LIN {X 0,Y 520,Z 902.665,A -85,B 0,C 180,E1 12177.794,E2 12177.794} C_VEL
LIN {X 0,Y 524.952,Z 869.378,A -85,B 0,C 180,E1 12181.307,E2 12181.307} C_VEL
LIN {X 0,Y 530.595,Z 831.105,A -85,B 0,C 180,E1 12184.398,E2 12184.398} C_VEL
LIN {X 0,Y 536.264,Z 787.905,A -85,B 0,C 180,E1 12186.977,E2 12186.977} C_VEL
LIN {X 0,Y 540.929,Z 743.185,A -85,B 0,C 180,E1 12188.852,E2 12188.852} C_VEL
LIN {X 0,Y 544.188,Z 696.094,A -85,B 0,C 180,E1 12190.101,E2 12190.101} C_VEL
LIN {X 0,Y 544.022,Z 681.132,A -85,B 0,C 180,E1 12190.406,E2 12190.406} C_VEL
LIN {X 0,Y 507.953,Z 601.31,A -85,B 0,C 180,E1 12194.386,E2 12194.386} C_VEL
LIN {X 0,Y 507.831,Z 601.31,A -85,B 0,C 180,E1 12200.881,E2 12200.881} C_VEL
LIN {X 0,Y 507.959,Z 601.31,A -85,B 0,C 180,E1 12206.647,E2 12206.647} C_VEL
LIN {X 0,Y 508.168,Z 601.31,A -85,B 0,C 180,E1 12211.51,E2 12211.51} C_VEL
LIN {X 0,Y 508.405,Z 601.31,A -85,B 0,C 180,E1 12217.515,E2 12217.515} C_VEL
LIN {X 0,Y 508.487,Z 601.31,A -85,B 0,C 180,E1 12222.665,E2 12222.665} C_VEL
LIN {X 0,Y 508.666,Z 601.31,A -85,B 0,C 180,E1 12227.965,E2 12227.965} C_VEL
LIN {X 0,Y 508.95,Z 601.31,A -85,B 0,C 180,E1 12233.16,E2 12233.16} C_VEL
LIN {X 0,Y 509.131,Z 601.31,A -85,B 0,C 180,E1 12238.293,E2 12238.293} C_VEL
LIN {X 0,Y 509.118,Z 601.31,A -85,B 0,C 180,E1 12243.41,E2 12243.41} C_VEL
LIN {X 0,Y 508.825,Z 601.31,A -85,B 0,C 180,E1 12248.559,E2 12248.559} C_VEL
LIN {X 0,Y 508.651,Z 601.31,A -85,B 0,C 180,E1 12253.782,E2 12253.782} C_VEL
LIN {X 0,Y 508.481,Z 601.31,A -85,B 0,C 180,E1 12259.128,E2 12259.128} C_VEL
LIN {X 0,Y 508.251,Z 601.31,A -85,B 0,C 180,E1 12264.661,E2 12264.661} C_VEL
LIN {X 0,Y 508.106,Z 601.31,A -85,B 0,C 180,E1 12270.451,E2 12270.451} C_VEL
LIN {X 0,Y 507.956,Z 601.31,A -85,B 0,C 180,E1 12276.614,E2 12276.614} C_VEL
LIN {X 0,Y 507.883,Z 601.31,A -85,B 0,C 180,E1 12283.314,E2 12283.314} C_VEL
LIN {X 0,Y 507.816,Z 601.31,A -85,B 0,C 180,E1 12288.966,E2 12288.966} C_VEL
LIN {X 0,Y 508.01,Z 601.31,A -85,B 0,C 180,E1 12295.314,E2 12295.314} C_VEL
LIN {X 0,Y 528.495,Z 651.414,A -85,B 0,C 180,E1 12298.224,E2 12298.224} C_VEL
LIN {X 0,Y 532.04,Z 668.727,A -85,B 0,C 180,E1 12299.099,E2 12299.099} C_VEL
LIN {X 0,Y 528.891,Z 707.618,A -85,B 0,C 180,E1 12300.849,E2 12300.849} C_VEL
LIN {X 0,Y 525.082,Z 743.156,A -85,B 0,C 180,E1 12303.155,E2 12303.155} C_VEL
LIN {X 0,Y 521.047,Z 775.217,A -85,B 0,C 180,E1 12305.971,E2 12305.971} C_VEL
LIN {X 0,Y 517.204,Z 804.444,A -85,B 0,C 180,E1 12309.413,E2 12309.413} C_VEL
LIN {X 0,Y 514.215,Z 827.771,A -85,B 0,C 180,E1 12313.102,E2 12313.102} C_VEL
LIN {X 0,Y 512.171,Z 846.045,A -85,B 0,C 180,E1 12317.034,E2 12317.034} C_VEL
LIN {X 0,Y 511.03,Z 859.031,A -85,B 0,C 180,E1 12321.04,E2 12321.04} C_VEL
LIN {X 0,Y 510.473,Z 866.812,A -85,B 0,C 180,E1 12324.887,E2 12324.887} C_VEL
LIN {X 0,Y 510.207,Z 870.137,A -85,B 0,C 180,E1 12328.294,E2 12328.294} C_VEL
LIN {X 0,Y 510.347,Z 870.07,A -85,B 0,C 180,E1 12331.697,E2 12331.697} C_VEL
LIN {X 0,Y 510.589,Z 865.782,A -85,B 0,C 180,E1 12335.703,E2 12335.703} C_VEL
LIN {X 0,Y 511.119,Z 856.498,A -85,B 0,C 180,E1 12339.81,E2 12339.81} C_VEL
LIN {X 0,Y 512.543,Z 842.831,A -85,B 0,C 180,E1 12343.675,E2 12343.675} C_VEL
LIN {X 0,Y 514.927,Z 822.28,A -85,B 0,C 180,E1 12347.771,E2 12347.771} C_VEL
LIN {X 0,Y 518.198,Z 797.24,A -85,B 0,C 180,E1 12351.433,E2 12351.433} C_VEL
LIN {X 0,Y 522.167,Z 766.734,A -85,B 0,C 180,E1 12354.763,E2 12354.763} C_VEL
LIN {X 0,Y 526.179,Z 733.773,A -85,B 0,C 180,E1 12357.43,E2 12357.43} C_VEL
LIN {X 0,Y 529.775,Z 697.922,A -85,B 0,C 180,E1 12359.557,E2 12359.557} C_VEL
LIN {X 0,Y 531.526,Z 665.249,A -85,B 0,C 180,E1 12360.976,E2 12360.976} C_VEL
LIN {X 0,Y 524.161,Z 639.669,A -85,B 0,C 180,E1 12362.329,E2 12362.329} C_VEL
LIN {X 0,Y 508.103,Z 601.31,A -85,B 0,C 180,E1 12364.601,E2 12364.601} C_VEL
LIN {X 0,Y 507.864,Z 601.31,A -85,B 0,C 180,E1 12371.017,E2 12371.017} C_VEL
LIN {X 0,Y 507.854,Z 601.31,A -85,B 0,C 180,E1 12376.683,E2 12376.683} C_VEL
LIN {X 0,Y 507.918,Z 601.31,A -85,B 0,C 180,E1 12383.383,E2 12383.383} C_VEL
LIN {X 0,Y 508.13,Z 601.31,A -85,B 0,C 180,E1 12389.846,E2 12389.846} C_VEL
LIN {X 0,Y 508.314,Z 601.31,A -85,B 0,C 180,E1 12394.173,E2 12394.173} C_VEL
LIN {X 0,Y 524.583,Z 651.894,A -85,B 0,C 180,E1 12395.94,E2 12395.94} C_VEL
LIN {X 0,Y 522.857,Z 701.074,A -85,B 0,C 180,E1 12396.974,E2 12396.974} C_VEL
LIN {X 0,Y 520.724,Z 738.628,A -85,B 0,C 180,E1 12398.437,E2 12398.437} C_VEL
LIN {X 0,Y 518.128,Z 773.015,A -85,B 0,C 180,E1 12400.466,E2 12400.466} C_VEL
LIN {X 0,Y 515.733,Z 803.731,A -85,B 0,C 180,E1 12403.031,E2 12403.031} C_VEL
LIN {X 0,Y 513.615,Z 830.564,A -85,B 0,C 180,E1 12406.137,E2 12406.137} C_VEL
LIN {X 0,Y 512.062,Z 851.637,A -85,B 0,C 180,E1 12409.562,E2 12409.562} C_VEL
LIN {X 0,Y 511.289,Z 866.871,A -85,B 0,C 180,E1 12413.196,E2 12413.196} C_VEL
LIN {X 0,Y 511.021,Z 875.647,A -85,B 0,C 180,E1 12416.603,E2 12416.603} C_VEL
LIN {X 0,Y 511.016,Z 879.604,A -85,B 0,C 180,E1 12420.002,E2 12420.002} C_VEL
LIN {X 0,Y 511.336,Z 878.832,A -85,B 0,C 180,E1 12423.399,E2 12423.399} C_VEL
LIN {X 0,Y 512.187,Z 873.073,A -85,B 0,C 180,E1 12426.797,E2 12426.797} C_VEL
LIN {X 0,Y 513.564,Z 862.006,A -85,B 0,C 180,E1 12430.196,E2 12430.196} C_VEL
LIN {X 0,Y 515.523,Z 844.762,A -85,B 0,C 180,E1 12433.599,E2 12433.599} C_VEL
LIN {X 0,Y 517.943,Z 822.966,A -85,B 0,C 180,E1 12436.571,E2 12436.571} C_VEL
LIN {X 0,Y 520.985,Z 794.562,A -85,B 0,C 180,E1 12439.378,E2 12439.378} C_VEL
LIN {X 0,Y 524.438,Z 759.753,A -85,B 0,C 180,E1 12441.835,E2 12441.835} C_VEL
LIN {X 0,Y 528.068,Z 719.982,A -85,B 0,C 180,E1 12443.78,E2 12443.78} C_VEL
LIN {X 0,Y 531.717,Z 674.928,A -85,B 0,C 180,E1 12445.188,E2 12445.188} C_VEL
LIN {X 0,Y 532.545,Z 655.359,A -85,B 0,C 180,E1 12445.707,E2 12445.707} C_VEL
LIN {X 0,Y 523.124,Z 630.3,A -85,B 0,C 180,E1 12447.507,E2 12447.507} C_VEL
LIN {X 0,Y 513.846,Z 612.495,A -85,B 0,C 180,E1 12449.435,E2 12449.435} C_VEL
LIN {X 0,Y 510.034,Z 606.45,A -85,B 0,C 180,E1 12450.329,E2 12450.329} C_VEL
LIN {X 0,Y 508.092,Z 601.31,A -85,B 0,C 180,E1 12451.036,E2 12451.036} C_VEL
LIN {X 0,Y 508,Z 601.31,A -85,B 0,C 180,E1 12456.616,E2 12456.616} C_VEL
LIN {X 0,Y 507.909,Z 601.31,A -85,B 0,C 180,E1 12463.317,E2 12463.317} C_VEL
LIN {X 0,Y 507.889,Z 601.868,A -85,B 0,C 180,E1 12464.024,E2 12464.024} C_VEL
LIN {X 0,Y 510.593,Z 607.203,A -85,B 0,C 180,E1 12464.707,E2 12464.707} C_VEL
LIN {X 0,Y 519.408,Z 621.579,A -85,B 0,C 180,E1 12466.437,E2 12466.437} C_VEL
LIN {X 0,Y 530.121,Z 643.576,A -85,B 0,C 180,E1 12468.173,E2 12468.173} C_VEL
LIN {X 0,Y 538.662,Z 670.296,A -85,B 0,C 180,E1 12469.492,E2 12469.492} C_VEL
LIN {X 0,Y 542.514,Z 685.222,A -85,B 0,C 180,E1 12470.096,E2 12470.096} C_VEL
LIN {X 0,Y 539.64,Z 730.719,A -85,B 0,C 180,E1 12471.16,E2 12471.16} C_VEL
LIN {X 0,Y 535.552,Z 773.807,A -85,B 0,C 180,E1 12472.795,E2 12472.795} C_VEL
LIN {X 0,Y 530.748,Z 816.248,A -85,B 0,C 180,E1 12475.111,E2 12475.111} C_VEL
LIN {X 0,Y 525.549,Z 855.463,A -85,B 0,C 180,E1 12477.983,E2 12477.983} C_VEL
LIN {X 0,Y 524.944,Z 859.637,A -85,B 0,C 180,E1 12478.346,E2 12478.346} C_VEL
LIN {X 0,Y 519.28,Z 873.172,A -85,B 0,C 180,E1 12479.413,E2 12479.413} C_VEL
LIN {X 0,Y 513.783,Z 886.061,A -85,B 0,C 180,E1 12480.57,E2 12480.57} C_VEL
LIN {X 0,Y 509.18,Z 917.936,A -85,B 0,C 180,E1 12484.443,E2 12484.443} C_VEL
LIN {X 0,Y 505.687,Z 945.186,A -85,B 0,C 180,E1 12488.724,E2 12488.724} C_VEL
LIN {X 0,Y 503.449,Z 967.671,A -85,B 0,C 180,E1 12493.391,E2 12493.391} C_VEL
LIN {X 0,Y 502.283,Z 984.168,A -85,B 0,C 180,E1 12498.167,E2 12498.167} C_VEL
LIN {X 0,Y 501.854,Z 993.668,A -85,B 0,C 180,E1 12502.196,E2 12502.196} C_VEL
LIN {X 0,Y 501.774,Z 999.535,A -85,B 0,C 180,E1 12506.542,E2 12506.542} C_VEL
LIN {X 0,Y 501.842,Z 1001.106,A -85,B 0,C 180,E1 12510.005,E2 12510.005} C_VEL
LIN {X 0,Y 501.849,Z 998.33,A -85,B 0,C 180,E1 12515.012,E2 12515.012} C_VEL
LIN {X 0,Y 501.97,Z 989.857,A -85,B 0,C 180,E1 12520,E2 12520} C_VEL
LIN {X 0,Y 502.842,Z 976.424,A -85,B 0,C 180,E1 12524.732,E2 12524.732} C_VEL
LIN {X 0,Y 504.859,Z 955.712,A -85,B 0,C 180,E1 12529.738,E2 12529.738} C_VEL
LIN {X 0,Y 508.329,Z 929.158,A -85,B 0,C 180,E1 12534.435,E2 12534.435} C_VEL
LIN {X 0,Y 512.81,Z 899.389,A -85,B 0,C 180,E1 12538.438,E2 12538.438} C_VEL
LIN {X 0,Y 518.058,Z 865.903,A -85,B 0,C 180,E1 12541.928,E2 12541.928} C_VEL
LIN {X 0,Y 523.721,Z 828.076,A -85,B 0,C 180,E1 12544.955,E2 12544.955} C_VEL
LIN {X 0,Y 529.236,Z 787.2,A -85,B 0,C 180,E1 12547.397,E2 12547.397} C_VEL
LIN {X 0,Y 534.129,Z 741.814,A -85,B 0,C 180,E1 12549.31,E2 12549.31} C_VEL
LIN {X 0,Y 537.459,Z 694.943,A -85,B 0,C 180,E1 12550.55,E2 12550.55} C_VEL
LIN {X 0,Y 537.203,Z 683.382,A -85,B 0,C 180,E1 12550.795,E2 12550.795} C_VEL
LIN {X 0,Y 500.024,Z 601.31,A -85,B 0,C 180,E1 12554.978,E2 12554.978} C_VEL
LIN {X 0,Y 499.903,Z 601.31,A -85,B 0,C 180,E1 12560.475,E2 12560.475} C_VEL
LIN {X 0,Y 500.061,Z 601.31,A -85,B 0,C 180,E1 12566.953,E2 12566.953} C_VEL
LIN {X 0,Y 500.242,Z 601.31,A -85,B 0,C 180,E1 12572.981,E2 12572.981} C_VEL
LIN {X 0,Y 500.476,Z 601.31,A -85,B 0,C 180,E1 12578.699,E2 12578.699} C_VEL
LIN {X 0,Y 500.619,Z 601.31,A -85,B 0,C 180,E1 12584.194,E2 12584.194} C_VEL
LIN {X 0,Y 500.847,Z 601.31,A -85,B 0,C 180,E1 12589.542,E2 12589.542} C_VEL
LIN {X 0,Y 501.148,Z 601.31,A -85,B 0,C 180,E1 12594.795,E2 12594.795} C_VEL
LIN {X 0,Y 501.325,Z 601.31,A -85,B 0,C 180,E1 12599.998,E2 12599.998} C_VEL
LIN {X 0,Y 501.177,Z 601.31,A -85,B 0,C 180,E1 12605.201,E2 12605.201} C_VEL
LIN {X 0,Y 500.866,Z 601.31,A -85,B 0,C 180,E1 12610.453,E2 12610.453} C_VEL
LIN {X 0,Y 500.654,Z 601.31,A -85,B 0,C 180,E1 12615.8,E2 12615.8} C_VEL
LIN {X 0,Y 500.499,Z 601.31,A -85,B 0,C 180,E1 12621.295,E2 12621.295} C_VEL
LIN {X 0,Y 500.227,Z 601.31,A -85,B 0,C 180,E1 12627.015,E2 12627.015} C_VEL
LIN {X 0,Y 500.08,Z 601.31,A -85,B 0,C 180,E1 12633.041,E2 12633.041} C_VEL
LIN {X 0,Y 499.942,Z 601.31,A -85,B 0,C 180,E1 12639.515,E2 12639.515} C_VEL
LIN {X 0,Y 499.975,Z 601.31,A -85,B 0,C 180,E1 12645.804,E2 12645.804} C_VEL
LIN {X 0,Y 499.894,Z 601.31,A -85,B 0,C 180,E1 12651.987,E2 12651.987} C_VEL
LIN {X 0,Y 500.05,Z 601.31,A -85,B 0,C 180,E1 12654.652,E2 12654.652} C_VEL
LIN {X 0,Y 520.969,Z 651.493,A -85,B 0,C 180,E1 12657.696,E2 12657.696} C_VEL
LIN {X 0,Y 525.141,Z 671.855,A -85,B 0,C 180,E1 12658.754,E2 12658.754} C_VEL
LIN {X 0,Y 521.749,Z 710.935,A -85,B 0,C 180,E1 12660.575,E2 12660.575} C_VEL
LIN {X 0,Y 517.831,Z 745.962,A -85,B 0,C 180,E1 12662.916,E2 12662.916} C_VEL
LIN {X 0,Y 513.605,Z 778.182,A -85,B 0,C 180,E1 12665.827,E2 12665.827} C_VEL
LIN {X 0,Y 509.516,Z 807.297,A -85,B 0,C 180,E1 12669.376,E2 12669.376} C_VEL
LIN {X 0,Y 506.449,Z 830.412,A -85,B 0,C 180,E1 12673.165,E2 12673.165} C_VEL
LIN {X 0,Y 504.3,Z 848.89,A -85,B 0,C 180,E1 12677.322,E2 12677.322} C_VEL
LIN {X 0,Y 503.139,Z 861.13,A -85,B 0,C 180,E1 12681.335,E2 12681.335} C_VEL
LIN {X 0,Y 502.601,Z 868.987,A -85,B 0,C 180,E1 12685.673,E2 12685.673} C_VEL
LIN {X 0,Y 502.513,Z 871.538,A -85,B 0,C 180,E1 12689.995,E2 12689.995} C_VEL
LIN {X 0,Y 502.633,Z 868.872,A -85,B 0,C 180,E1 12694.317,E2 12694.317} C_VEL
LIN {X 0,Y 503.231,Z 860.902,A -85,B 0,C 180,E1 12698.654,E2 12698.654} C_VEL
LIN {X 0,Y 504.5,Z 847.214,A -85,B 0,C 180,E1 12703.016,E2 12703.016} C_VEL
LIN {X 0,Y 506.733,Z 828.038,A -85,B 0,C 180,E1 12707.19,E2 12707.19} C_VEL
LIN {X 0,Y 510.106,Z 803.151,A -85,B 0,C 180,E1 12711.105,E2 12711.105} C_VEL
LIN {X 0,Y 514.092,Z 774.214,A -85,B 0,C 180,E1 12714.481,E2 12714.481} C_VEL
LIN {X 0,Y 518.385,Z 741.285,A -85,B 0,C 180,E1 12717.351,E2 12717.351} C_VEL
LIN {X 0,Y 522.276,Z 705.207,A -85,B 0,C 180,E1 12719.645,E2 12719.645} C_VEL
LIN {X 0,Y 524.671,Z 667.194,A -85,B 0,C 180,E1 12721.37,E2 12721.37} C_VEL
LIN {X 0,Y 517.609,Z 642.557,A -85,B 0,C 180,E1 12722.713,E2 12722.713} C_VEL
LIN {X 0,Y 500.132,Z 601.31,A -85,B 0,C 180,E1 12725.243,E2 12725.243} C_VEL
LIN {X 0,Y 499.999,Z 601.31,A -85,B 0,C 180,E1 12731.806,E2 12731.806} C_VEL
LIN {X 0,Y 499.941,Z 601.31,A -85,B 0,C 180,E1 12738.196,E2 12738.196} C_VEL
LIN {X 0,Y 500.033,Z 601.31,A -85,B 0,C 180,E1 12744.892,E2 12744.892} C_VEL
LIN {X 0,Y 500.249,Z 601.31,A -85,B 0,C 180,E1 12751.438,E2 12751.438} C_VEL
LIN {X 0,Y 500.361,Z 601.31,A -85,B 0,C 180,E1 12753.777,E2 12753.777} C_VEL
LIN {X 0,Y 517.186,Z 655.212,A -85,B 0,C 180,E1 12755.678,E2 12755.678} C_VEL
LIN {X 0,Y 515.422,Z 701.486,A -85,B 0,C 180,E1 12756.683,E2 12756.683} C_VEL
LIN {X 0,Y 513.224,Z 738.97,A -85,B 0,C 180,E1 12758.166,E2 12758.166} C_VEL
LIN {X 0,Y 510.497,Z 774.133,A -85,B 0,C 180,E1 12760.275,E2 12760.275} C_VEL
LIN {X 0,Y 507.881,Z 805.823,A -85,B 0,C 180,E1 12762.984,E2 12762.984} C_VEL
LIN {X 0,Y 505.767,Z 832.36,A -85,B 0,C 180,E1 12766.138,E2 12766.138} C_VEL
LIN {X 0,Y 504.242,Z 853.261,A -85,B 0,C 180,E1 12769.618,E2 12769.618} C_VEL
LIN {X 0,Y 503.42,Z 868.26,A -85,B 0,C 180,E1 12773.293,E2 12773.293} C_VEL
LIN {X 0,Y 503.198,Z 876.534,A -85,B 0,C 180,E1 12776.55,E2 12776.55} C_VEL
LIN {X 0,Y 503.195,Z 880.651,A -85,B 0,C 180,E1 12780.002,E2 12780.002} C_VEL
LIN {X 0,Y 503.537,Z 880.006,A -85,B 0,C 180,E1 12783.452,E2 12783.452} C_VEL
LIN {X 0,Y 504.456,Z 874.408,A -85,B 0,C 180,E1 12786.901,E2 12786.901} C_VEL
LIN {X 0,Y 505.933,Z 863.428,A -85,B 0,C 180,E1 12790.352,E2 12790.352} C_VEL
LIN {X 0,Y 508.01,Z 846.33,A -85,B 0,C 180,E1 12793.804,E2 12793.804} C_VEL
LIN {X 0,Y 510.587,Z 824.772,A -85,B 0,C 180,E1 12796.817,E2 12796.817} C_VEL
LIN {X 0,Y 513.842,Z 796.322,A -85,B 0,C 180,E1 12799.696,E2 12799.696} C_VEL
LIN {X 0,Y 517.401,Z 762.529,A -85,B 0,C 180,E1 12802.148,E2 12802.148} C_VEL
LIN {X 0,Y 521.217,Z 723.88,A -85,B 0,C 180,E1 12804.127,E2 12804.127} C_VEL
LIN {X 0,Y 524.994,Z 682.276,A -85,B 0,C 180,E1 12805.535,E2 12805.535} C_VEL
LIN {X 0,Y 526.375,Z 657.824,A -85,B 0,C 180,E1 12806.206,E2 12806.206} C_VEL
LIN {X 0,Y 517.228,Z 633.141,A -85,B 0,C 180,E1 12808.099,E2 12808.099} C_VEL
LIN {X 0,Y 507.4,Z 614.083,A -85,B 0,C 180,E1 12810.387,E2 12810.387} C_VEL
LIN {X 0,Y 502.885,Z 607.264,A -85,B 0,C 180,E1 12811.64,E2 12811.64} C_VEL
LIN {X 0,Y 500.132,Z 601.853,A -85,B 0,C 180,E1 12812.655,E2 12812.655} C_VEL
LIN {X 0,Y 499.988,Z 601.31,A -85,B 0,C 180,E1 12818.016,E2 12818.016} C_VEL
LIN {X 0,Y 500.023,Z 601.976,A -85,B 0,C 180,E1 12822.293,E2 12822.293} C_VEL
LIN {X 0,Y 502.726,Z 607.254,A -85,B 0,C 180,E1 12823.217,E2 12823.217} C_VEL
LIN {X 0,Y 504.974,Z 610.344,A -85,B 0,C 180,E1 12823.816,E2 12823.816} C_VEL
LIN {X 0,Y 512.671,Z 622.71,A -85,B 0,C 180,E1 12825.547,E2 12825.547} C_VEL
LIN {X 0,Y 522.833,Z 642.836,A -85,B 0,C 180,E1 12827.38,E2 12827.38} C_VEL
LIN {X 0,Y 530.974,Z 666.365,A -85,B 0,C 180,E1 12828.724,E2 12828.724} C_VEL
LIN {X 0,Y 536.271,Z 685.119,A -85,B 0,C 180,E1 12829.578,E2 12829.578} C_VEL
LIN {X 0,Y 533.213,Z 730.537,A -85,B 0,C 180,E1 12830.665,E2 12830.665} C_VEL
LIN {X 0,Y 528.819,Z 773.973,A -85,B 0,C 180,E1 12832.345,E2 12832.345} C_VEL
LIN {X 0,Y 523.816,Z 815.666,A -85,B 0,C 180,E1 12834.659,E2 12834.659} C_VEL
LIN {X 0,Y 518.24,Z 855.553,A -85,B 0,C 180,E1 12837.635,E2 12837.635} C_VEL
LIN {X 0,Y 513.783,Z 886.061,A -85,B 0,C 180,E1 12840.57,E2 12840.57} C_VEL
LIN {X 0,Y 511.734,Z 892.403,A -85,B 0,C 180,E1 12841.213,E2 12841.213} C_VEL
LIN {X 0,Y 502.927,Z 908.748,A -85,B 0,C 180,E1 12842.967,E2 12842.967} C_VEL
LIN {X 0,Y 502.65,Z 910.185,A -85,B 0,C 180,E1 12843.151,E2 12843.151} C_VEL
LIN {X 0,Y 498.838,Z 937.618,A -85,B 0,C 180,E1 12847.266,E2 12847.266} C_VEL
LIN {X 0,Y 496.197,Z 960.3,A -85,B 0,C 180,E1 12851.654,E2 12851.654} C_VEL
LIN {X 0,Y 494.6,Z 979.493,A -85,B 0,C 180,E1 12856.722,E2 12856.722} C_VEL
LIN {X 0,Y 494.084,Z 990.97,A -85,B 0,C 180,E1 12861.185,E2 12861.185} C_VEL
LIN {X 0,Y 494.027,Z 996.816,A -85,B 0,C 180,E1 12864.726,E2 12864.726} C_VEL
LIN {X 0,Y 494.011,Z 999.798,A -85,B 0,C 180,E1 12868.247,E2 12868.247} C_VEL
LIN {X 0,Y 493.881,Z 999.942,A -85,B 0,C 180,E1 12871.763,E2 12871.763} C_VEL
LIN {X 0,Y 493.93,Z 996.144,A -85,B 0,C 180,E1 12876.168,E2 12876.168} C_VEL
LIN {X 0,Y 494.288,Z 986.415,A -85,B 0,C 180,E1 12881.256,E2 12881.256} C_VEL
LIN {X 0,Y 495.482,Z 970.106,A -85,B 0,C 180,E1 12886.437,E2 12886.437} C_VEL
LIN {X 0,Y 497.803,Z 948.823,A -85,B 0,C 180,E1 12891.194,E2 12891.194} C_VEL
LIN {X 0,Y 501.484,Z 923.247,A -85,B 0,C 180,E1 12895.508,E2 12895.508} C_VEL
LIN {X 0,Y 506.338,Z 892.85,A -85,B 0,C 180,E1 12899.464,E2 12899.464} C_VEL
LIN {X 0,Y 512.022,Z 857.355,A -85,B 0,C 180,E1 12903.018,E2 12903.018} C_VEL
LIN {X 0,Y 518.09,Z 816.765,A -85,B 0,C 180,E1 12906.085,E2 12906.085} C_VEL
LIN {X 0,Y 523.914,Z 771.768,A -85,B 0,C 180,E1 12908.538,E2 12908.538} C_VEL
LIN {X 0,Y 528.471,Z 726.177,A -85,B 0,C 180,E1 12910.225,E2 12910.225} C_VEL
LIN {X 0,Y 530.451,Z 685.946,A -85,B 0,C 180,E1 12911.175,E2 12911.175} C_VEL
LIN {X 0,Y 492.065,Z 601.31,A -85,B 0,C 180,E1 12915.556,E2 12915.556} C_VEL
LIN {X 0,Y 492.01,Z 601.31,A -85,B 0,C 180,E1 12921.988,E2 12921.988} C_VEL
LIN {X 0,Y 492.168,Z 601.31,A -85,B 0,C 180,E1 12928.447,E2 12928.447} C_VEL
LIN {X 0,Y 492.348,Z 601.31,A -85,B 0,C 180,E1 12934.482,E2 12934.482} C_VEL
LIN {X 0,Y 492.582,Z 601.31,A -85,B 0,C 180,E1 12940.225,E2 12940.225} C_VEL
LIN {X 0,Y 492.729,Z 601.31,A -85,B 0,C 180,E1 12945.759,E2 12945.759} C_VEL
LIN {X 0,Y 493.001,Z 601.31,A -85,B 0,C 180,E1 12951.16,E2 12951.16} C_VEL
LIN {X 0,Y 493.338,Z 601.31,A -85,B 0,C 180,E1 12956.477,E2 12956.477} C_VEL
LIN {X 0,Y 493.447,Z 601.31,A -85,B 0,C 180,E1 12961.757,E2 12961.757} C_VEL
LIN {X 0,Y 493.111,Z 601.31,A -85,B 0,C 180,E1 12967.056,E2 12967.056} C_VEL
LIN {X 0,Y 492.847,Z 601.31,A -85,B 0,C 180,E1 12972.423,E2 12972.423} C_VEL
LIN {X 0,Y 492.667,Z 601.31,A -85,B 0,C 180,E1 12977.905,E2 12977.905} C_VEL
LIN {X 0,Y 492.444,Z 601.31,A -85,B 0,C 180,E1 12983.57,E2 12983.57} C_VEL
LIN {X 0,Y 492.227,Z 601.31,A -85,B 0,C 180,E1 12989.497,E2 12989.497} C_VEL
LIN {X 0,Y 492.058,Z 601.31,A -85,B 0,C 180,E1 12995.796,E2 12995.796} C_VEL
LIN {X 0,Y 492.059,Z 601.31,A -85,B 0,C 180,E1 13002.343,E2 13002.343} C_VEL
LIN {X 0,Y 492.036,Z 601.31,A -85,B 0,C 180,E1 13007.636,E2 13007.636} C_VEL
LIN {X 0,Y 492.167,Z 601.598,A -85,B 0,C 180,E1 13014.002,E2 13014.002} C_VEL
LIN {X 0,Y 513.135,Z 650.798,A -85,B 0,C 180,E1 13017.111,E2 13017.111} C_VEL
LIN {X 0,Y 518.412,Z 672.347,A -85,B 0,C 180,E1 13018.302,E2 13018.302} C_VEL
LIN {X 0,Y 514.926,Z 711.698,A -85,B 0,C 180,E1 13020.146,E2 13020.146} C_VEL
LIN {X 0,Y 510.696,Z 747.83,A -85,B 0,C 180,E1 13022.595,E2 13022.595} C_VEL
LIN {X 0,Y 506.301,Z 780.014,A -85,B 0,C 180,E1 13025.561,E2 13025.561} C_VEL
LIN {X 0,Y 502.029,Z 809.024,A -85,B 0,C 180,E1 13029.176,E2 13029.176} C_VEL
LIN {X 0,Y 498.707,Z 832.634,A -85,B 0,C 180,E1 13033.147,E2 13033.147} C_VEL
LIN {X 0,Y 496.459,Z 851.295,A -85,B 0,C 180,E1 13037.528,E2 13037.528} C_VEL
LIN {X 0,Y 495.221,Z 864.071,A -85,B 0,C 180,E1 13042.081,E2 13042.081} C_VEL
LIN {X 0,Y 494.684,Z 870.844,A -85,B 0,C 180,E1 13046.483,E2 13046.483} C_VEL
LIN {X 0,Y 494.675,Z 872.526,A -85,B 0,C 180,E1 13049.995,E2 13049.995} C_VEL
LIN {X 0,Y 494.813,Z 869.855,A -85,B 0,C 180,E1 13054.386,E2 13054.386} C_VEL
LIN {X 0,Y 495.451,Z 861.878,A -85,B 0,C 180,E1 13058.791,E2 13058.791} C_VEL
LIN {X 0,Y 496.831,Z 848.192,A -85,B 0,C 180,E1 13063.216,E2 13063.216} C_VEL
LIN {X 0,Y 499.153,Z 829.396,A -85,B 0,C 180,E1 13067.38,E2 13067.38} C_VEL
LIN {X 0,Y 502.767,Z 804.065,A -85,B 0,C 180,E1 13071.428,E2 13071.428} C_VEL
LIN {X 0,Y 506.928,Z 775.109,A -85,B 0,C 180,E1 13074.85,E2 13074.85} C_VEL
LIN {X 0,Y 511.48,Z 741.669,A -85,B 0,C 180,E1 13077.792,E2 13077.792} C_VEL
LIN {X 0,Y 515.585,Z 704.541,A -85,B 0,C 180,E1 13080.15,E2 13080.15} C_VEL
LIN {X 0,Y 517.838,Z 669.07,A -85,B 0,C 180,E1 13081.776,E2 13081.776} C_VEL
LIN {X 0,Y 510.746,Z 644.586,A -85,B 0,C 180,E1 13083.158,E2 13083.158} C_VEL
LIN {X 0,Y 492.218,Z 601.31,A -85,B 0,C 180,E1 13085.917,E2 13085.917} C_VEL
LIN {X 0,Y 492.059,Z 601.31,A -85,B 0,C 180,E1 13092.638,E2 13092.638} C_VEL
LIN {X 0,Y 492.02,Z 601.31,A -85,B 0,C 180,E1 13097.647,E2 13097.647} C_VEL
LIN {X 0,Y 492.01,Z 601.31,A -85,B 0,C 180,E1 13104.2,E2 13104.2} C_VEL
LIN {X 0,Y 492.242,Z 601.31,A -85,B 0,C 180,E1 13110.504,E2 13110.504} C_VEL
LIN {X 0,Y 492.42,Z 601.31,A -85,B 0,C 180,E1 13113.362,E2 13113.362} C_VEL
LIN {X 0,Y 509.852,Z 655.963,A -85,B 0,C 180,E1 13115.367,E2 13115.367} C_VEL
LIN {X 0,Y 508.001,Z 702.075,A -85,B 0,C 180,E1 13116.389,E2 13116.389} C_VEL
LIN {X 0,Y 505.719,Z 739.812,A -85,B 0,C 180,E1 13117.913,E2 13117.913} C_VEL
LIN {X 0,Y 502.863,Z 775.24,A -85,B 0,C 180,E1 13120.077,E2 13120.077} C_VEL
LIN {X 0,Y 500.286,Z 806.05,A -85,B 0,C 180,E1 13122.746,E2 13122.746} C_VEL
LIN {X 0,Y 498.071,Z 832.625,A -85,B 0,C 180,E1 13125.92,E2 13125.92} C_VEL
LIN {X 0,Y 496.455,Z 853.767,A -85,B 0,C 180,E1 13129.453,E2 13129.453} C_VEL
LIN {X 0,Y 495.677,Z 868.314,A -85,B 0,C 180,E1 13132.98,E2 13132.98} C_VEL
LIN {X 0,Y 495.373,Z 877.429,A -85,B 0,C 180,E1 13136.496,E2 13136.496} C_VEL
LIN {X 0,Y 495.366,Z 881.699,A -85,B 0,C 180,E1 13140.002,E2 13140.002} C_VEL
LIN {X 0,Y 495.741,Z 881.191,A -85,B 0,C 180,E1 13143.506,E2 13143.506} C_VEL
LIN {X 0,Y 496.745,Z 875.739,A -85,B 0,C 180,E1 13147.009,E2 13147.009} C_VEL
LIN {X 0,Y 498.303,Z 864.915,A -85,B 0,C 180,E1 13150.512,E2 13150.512} C_VEL
LIN {X 0,Y 500.521,Z 847.972,A -85,B 0,C 180,E1 13154.014,E2 13154.014} C_VEL
LIN {X 0,Y 503.505,Z 824.841,A -85,B 0,C 180,E1 13157.286,E2 13157.286} C_VEL
LIN {X 0,Y 506.992,Z 795.99,A -85,B 0,C 180,E1 13160.214,E2 13160.214} C_VEL
LIN {X 0,Y 511.097,Z 760.341,A -85,B 0,C 180,E1 13162.793,E2 13162.793} C_VEL
LIN {X 0,Y 515.223,Z 721.295,A -85,B 0,C 180,E1 13164.773,E2 13164.773} C_VEL
LIN {X 0,Y 519.331,Z 678.345,A -85,B 0,C 180,E1 13166.21,E2 13166.21} C_VEL
LIN {X 0,Y 520.369,Z 660.306,A -85,B 0,C 180,E1 13166.736,E2 13166.736} C_VEL
LIN {X 0,Y 511.959,Z 637.259,A -85,B 0,C 180,E1 13168.61,E2 13168.61} C_VEL
LIN {X 0,Y 503.435,Z 620.256,A -85,B 0,C 180,E1 13170.769,E2 13170.769} C_VEL
LIN {X 0,Y 498.729,Z 613.018,A -85,B 0,C 180,E1 13172.215,E2 13172.215} C_VEL
LIN {X 0,Y 496.132,Z 608.125,A -85,B 0,C 180,E1 13173.297,E2 13173.297} C_VEL
LIN {X 0,Y 492.169,Z 602.151,A -85,B 0,C 180,E1 13175.759,E2 13175.759} C_VEL
LIN {X 0,Y 492.075,Z 601.654,A -85,B 0,C 180,E1 13179.032,E2 13179.032} C_VEL
LIN {X 0,Y 495.389,Z 607.746,A -85,B 0,C 180,E1 13181.301,E2 13181.301} C_VEL
LIN {X 0,Y 497.333,Z 609.914,A -85,B 0,C 180,E1 13182.04,E2 13182.04} C_VEL
LIN {X 0,Y 502.656,Z 618.608,A -85,B 0,C 180,E1 13183.712,E2 13183.712} C_VEL
LIN {X 0,Y 510.552,Z 631.664,A -85,B 0,C 180,E1 13185.511,E2 13185.511} C_VEL
LIN {X 0,Y 520.242,Z 653.231,A -85,B 0,C 180,E1 13187.331,E2 13187.331} C_VEL
LIN {X 0,Y 529.915,Z 686.896,A -85,B 0,C 180,E1 13189.055,E2 13189.055} C_VEL
LIN {X 0,Y 526.636,Z 732.845,A -85,B 0,C 180,E1 13190.223,E2 13190.223} C_VEL
LIN {X 0,Y 521.861,Z 776.603,A -85,B 0,C 180,E1 13191.991,E2 13191.991} C_VEL
LIN {X 0,Y 516.652,Z 817.297,A -85,B 0,C 180,E1 13194.335,E2 13194.335} C_VEL
LIN {X 0,Y 511.037,Z 855.396,A -85,B 0,C 180,E1 13197.247,E2 13197.247} C_VEL
LIN {X 0,Y 505.494,Z 891.768,A -85,B 0,C 180,E1 13200.886,E2 13200.886} C_VEL
LIN {X 0,Y 502.65,Z 910.185,A -85,B 0,C 180,E1 13203.151,E2 13203.151} C_VEL
LIN {X 0,Y 500.658,Z 915.879,A -85,B 0,C 180,E1 13203.879,E2 13203.879} C_VEL
LIN {X 0,Y 492.108,Z 930.466,A -85,B 0,C 180,E1 13205.889,E2 13205.889} C_VEL
LIN {X 0,Y 491.865,Z 931.76,A -85,B 0,C 180,E1 13206.093,E2 13206.093} C_VEL
LIN {X 0,Y 488.673,Z 956.569,A -85,B 0,C 180,E1 13210.777,E2 13210.777} C_VEL
LIN {X 0,Y 486.948,Z 975.488,A -85,B 0,C 180,E1 13215.591,E2 13215.591} C_VEL
LIN {X 0,Y 486.282,Z 988.134,A -85,B 0,C 180,E1 13220.137,E2 13220.137} C_VEL
LIN {X 0,Y 486.183,Z 995.909,A -85,B 0,C 180,E1 13224.64,E2 13224.64} C_VEL
LIN {X 0,Y 486.159,Z 998.914,A -85,B 0,C 180,E1 13228.219,E2 13228.219} C_VEL
LIN {X 0,Y 486.033,Z 999.074,A -85,B 0,C 180,E1 13231.791,E2 13231.791} C_VEL
LIN {X 0,Y 486.063,Z 995.249,A -85,B 0,C 180,E1 13236.269,E2 13236.269} C_VEL
LIN {X 0,Y 486.417,Z 985.462,A -85,B 0,C 180,E1 13241.44,E2 13241.44} C_VEL
LIN {X 0,Y 487.659,Z 969.038,A -85,B 0,C 180,E1 13246.708,E2 13246.708} C_VEL
LIN {X 0,Y 490.135,Z 947.596,A -85,B 0,C 180,E1 13251.542,E2 13251.542} C_VEL
LIN {X 0,Y 494.016,Z 921.782,A -85,B 0,C 180,E1 13255.922,E2 13255.922} C_VEL
LIN {X 0,Y 498.937,Z 891.624,A -85,B 0,C 180,E1 13259.871,E2 13259.871} C_VEL
LIN {X 0,Y 504.887,Z 855.882,A -85,B 0,C 180,E1 13263.472,E2 13263.472} C_VEL
LIN {X 0,Y 511.123,Z 815.171,A -85,B 0,C 180,E1 13266.553,E2 13266.553} C_VEL
LIN {X 0,Y 516.91,Z 771.703,A -85,B 0,C 180,E1 13268.945,E2 13268.945} C_VEL
LIN {X 0,Y 521.704,Z 724.989,A -85,B 0,C 180,E1 13270.685,E2 13270.685} C_VEL
LIN {X 0,Y 523.8,Z 688.696,A -85,B 0,C 180,E1 13271.551,E2 13271.551} C_VEL
LIN {X 0,Y 485.425,Z 605.588,A -85,B 0,C 180,E1 13275.906,E2 13275.906} C_VEL
LIN {X 0,Y 484.14,Z 601.31,A -85,B 0,C 180,E1 13276.112,E2 13276.112} C_VEL
LIN {X 0,Y 484.064,Z 601.31,A -85,B 0,C 180,E1 13281.502,E2 13281.502} C_VEL
LIN {X 0,Y 484.175,Z 601.31,A -85,B 0,C 180,E1 13287.864,E2 13287.864} C_VEL
LIN {X 0,Y 484.412,Z 601.31,A -85,B 0,C 180,E1 13294.033,E2 13294.033} C_VEL
LIN {X 0,Y 484.631,Z 601.31,A -85,B 0,C 180,E1 13299.886,E2 13299.886} C_VEL
LIN {X 0,Y 484.824,Z 601.31,A -85,B 0,C 180,E1 13305.677,E2 13305.677} C_VEL
LIN {X 0,Y 485.084,Z 601.31,A -85,B 0,C 180,E1 13311.014,E2 13311.014} C_VEL
LIN {X 0,Y 485.429,Z 601.31,A -85,B 0,C 180,E1 13316.419,E2 13316.419} C_VEL
LIN {X 0,Y 485.541,Z 601.31,A -85,B 0,C 180,E1 13321.786,E2 13321.786} C_VEL
LIN {X 0,Y 485.188,Z 601.31,A -85,B 0,C 180,E1 13327.172,E2 13327.172} C_VEL
LIN {X 0,Y 484.919,Z 601.31,A -85,B 0,C 180,E1 13332.629,E2 13332.629} C_VEL
LIN {X 0,Y 484.72,Z 601.31,A -85,B 0,C 180,E1 13338.209,E2 13338.209} C_VEL
LIN {X 0,Y 484.474,Z 601.31,A -85,B 0,C 180,E1 13343.982,E2 13343.982} C_VEL
LIN {X 0,Y 484.292,Z 601.31,A -85,B 0,C 180,E1 13350.029,E2 13350.029} C_VEL
LIN {X 0,Y 484.12,Z 601.31,A -85,B 0,C 180,E1 13356.477,E2 13356.477} C_VEL
LIN {X 0,Y 484.072,Z 601.31,A -85,B 0,C 180,E1 13361.296,E2 13361.296} C_VEL
LIN {X 0,Y 484.046,Z 601.31,A -85,B 0,C 180,E1 13366.469,E2 13366.469} C_VEL
LIN {X 0,Y 484.175,Z 601.31,A -85,B 0,C 180,E1 13373.242,E2 13373.242} C_VEL
LIN {X 0,Y 505.554,Z 650.75,A -85,B 0,C 180,E1 13376.542,E2 13376.542} C_VEL
LIN {X 0,Y 511.693,Z 673.462,A -85,B 0,C 180,E1 13377.862,E2 13377.862} C_VEL
LIN {X 0,Y 508.086,Z 712.755,A -85,B 0,C 180,E1 13379.721,E2 13379.721} C_VEL
LIN {X 0,Y 503.706,Z 748.879,A -85,B 0,C 180,E1 13382.2,E2 13382.2} C_VEL
LIN {X 0,Y 498.951,Z 782.264,A -85,B 0,C 180,E1 13385.336,E2 13385.336} C_VEL
LIN {X 0,Y 494.812,Z 809.141,A -85,B 0,C 180,E1 13388.731,E2 13388.731} C_VEL
LIN {X 0,Y 491.376,Z 832.348,A -85,B 0,C 180,E1 13392.641,E2 13392.641} C_VEL
LIN {X 0,Y 488.912,Z 851.155,A -85,B 0,C 180,E1 13397.011,E2 13397.011} C_VEL
LIN {X 0,Y 487.628,Z 863.073,A -85,B 0,C 180,E1 13401.057,E2 13401.057} C_VEL
LIN {X 0,Y 486.974,Z 870.951,A -85,B 0,C 180,E1 13405.534,E2 13405.534} C_VEL
LIN {X 0,Y 486.853,Z 873.512,A -85,B 0,C 180,E1 13409.995,E2 13409.995} C_VEL
LIN {X 0,Y 487.003,Z 870.838,A -85,B 0,C 180,E1 13414.456,E2 13414.456} C_VEL
LIN {X 0,Y 487.665,Z 862.858,A -85,B 0,C 180,E1 13418.932,E2 13418.932} C_VEL
LIN {X 0,Y 489.17,Z 849.157,A -85,B 0,C 180,E1 13423.428,E2 13423.428} C_VEL
LIN {X 0,Y 491.62,Z 830.399,A -85,B 0,C 180,E1 13427.647,E2 13427.647} C_VEL
LIN {X 0,Y 495.439,Z 804.992,A -85,B 0,C 180,E1 13431.761,E2 13431.761} C_VEL
LIN {X 0,Y 499.805,Z 776.011,A -85,B 0,C 180,E1 13435.229,E2 13435.229} C_VEL
LIN {X 0,Y 504.543,Z 742.482,A -85,B 0,C 180,E1 13438.209,E2 13438.209} C_VEL
LIN {X 0,Y 508.658,Z 706.803,A -85,B 0,C 180,E1 13440.513,E2 13440.513} C_VEL
LIN {X 0,Y 511.086,Z 671.219,A -85,B 0,C 180,E1 13442.179,E2 13442.179} C_VEL
LIN {X 0,Y 504.091,Z 647.121,A -85,B 0,C 180,E1 13443.585,E2 13443.585} C_VEL
LIN {X 0,Y 485.517,Z 605.549,A -85,B 0,C 180,E1 13446.372,E2 13446.372} C_VEL
LIN {X 0,Y 484.251,Z 601.31,A -85,B 0,C 180,E1 13446.653,E2 13446.653} C_VEL
LIN {X 0,Y 484.062,Z 601.31,A -85,B 0,C 180,E1 13453.516,E2 13453.516} C_VEL
LIN {X 0,Y 484.036,Z 601.31,A -85,B 0,C 180,E1 13458.914,E2 13458.914} C_VEL
LIN {X 0,Y 484.085,Z 601.31,A -85,B 0,C 180,E1 13464.461,E2 13464.461} C_VEL
LIN {X 0,Y 484.315,Z 601.31,A -85,B 0,C 180,E1 13471.153,E2 13471.153} C_VEL
LIN {X 0,Y 484.524,Z 601.607,A -85,B 0,C 180,E1 13472.963,E2 13472.963} C_VEL
LIN {X 0,Y 502.429,Z 656.37,A -85,B 0,C 180,E1 13475.034,E2 13475.034} C_VEL
LIN {X 0,Y 500.602,Z 702.343,A -85,B 0,C 180,E1 13476.076,E2 13476.076} C_VEL
LIN {X 0,Y 498.18,Z 740.87,A -85,B 0,C 180,E1 13477.662,E2 13477.662} C_VEL
LIN {X 0,Y 495.246,Z 776.343,A -85,B 0,C 180,E1 13479.874,E2 13479.874} C_VEL
LIN {X 0,Y 492.575,Z 807.185,A -85,B 0,C 180,E1 13482.595,E2 13482.595} C_VEL
LIN {X 0,Y 490.265,Z 833.878,A -85,B 0,C 180,E1 13485.842,E2 13485.842} C_VEL
LIN {X 0,Y 488.606,Z 855.354,A -85,B 0,C 180,E1 13489.507,E2 13489.507} C_VEL
LIN {X 0,Y 487.754,Z 870.506,A -85,B 0,C 180,E1 13493.334,E2 13493.334} C_VEL
LIN {X 0,Y 487.537,Z 879.863,A -85,B 0,C 180,E1 13497.331,E2 13497.331} C_VEL
LIN {X 0,Y 487.545,Z 882.73,A -85,B 0,C 180,E1 13500.002,E2 13500.002} C_VEL
LIN {X 0,Y 487.969,Z 882.381,A -85,B 0,C 180,E1 13503.562,E2 13503.562} C_VEL
LIN {X 0,Y 489.015,Z 877.089,A -85,B 0,C 180,E1 13507.12,E2 13507.12} C_VEL
LIN {X 0,Y 490.705,Z 866.406,A -85,B 0,C 180,E1 13510.677,E2 13510.677} C_VEL
LIN {X 0,Y 493.036,Z 849.638,A -85,B 0,C 180,E1 13514.232,E2 13514.232} C_VEL
LIN {X 0,Y 496.21,Z 826.825,A -85,B 0,C 180,E1 13517.548,E2 13517.548} C_VEL
LIN {X 0,Y 499.905,Z 798.451,A -85,B 0,C 180,E1 13520.512,E2 13520.512} C_VEL
LIN {X 0,Y 504.174,Z 763.719,A -85,B 0,C 180,E1 13523.124,E2 13523.124} C_VEL
LIN {X 0,Y 508.754,Z 723.999,A -85,B 0,C 180,E1 13525.227,E2 13525.227} C_VEL
LIN {X 0,Y 513.491,Z 678.993,A -85,B 0,C 180,E1 13526.795,E2 13526.795} C_VEL
LIN {X 0,Y 514.401,Z 662.647,A -85,B 0,C 180,E1 13527.296,E2 13527.296} C_VEL
LIN {X 0,Y 506.419,Z 640.139,A -85,B 0,C 180,E1 13529.27,E2 13529.27} C_VEL
LIN {X 0,Y 498.735,Z 625.01,A -85,B 0,C 180,E1 13531.431,E2 13531.431} C_VEL
LIN {X 0,Y 493.356,Z 615.375,A -85,B 0,C 180,E1 13533.555,E2 13533.555} C_VEL
LIN {X 0,Y 489.751,Z 608.855,A -85,B 0,C 180,E1 13536.456,E2 13536.456} C_VEL
LIN {X 0,Y 490.096,Z 609.71,A -85,B 0,C 180,E1 13538.966,E2 13538.966} C_VEL
LIN {X 0,Y 493.959,Z 615.67,A -85,B 0,C 180,E1 13541.418,E2 13541.418} C_VEL
LIN {X 0,Y 501.482,Z 627.884,A -85,B 0,C 180,E1 13543.869,E2 13543.869} C_VEL
LIN {X 0,Y 510.62,Z 646.007,A -85,B 0,C 180,E1 13545.945,E2 13545.945} C_VEL
LIN {X 0,Y 518.34,Z 667.397,A -85,B 0,C 180,E1 13547.447,E2 13547.447} C_VEL
LIN {X 0,Y 523.94,Z 690.75,A -85,B 0,C 180,E1 13548.579,E2 13548.579} C_VEL
LIN {X 0,Y 519.693,Z 739.492,A -85,B 0,C 180,E1 13549.908,E2 13549.908} C_VEL
LIN {X 0,Y 514.277,Z 784.544,A -85,B 0,C 180,E1 13551.893,E2 13551.893} C_VEL
LIN {X 0,Y 508.245,Z 826.994,A -85,B 0,C 180,E1 13554.552,E2 13554.552} C_VEL
LIN {X 0,Y 502.176,Z 865.769,A -85,B 0,C 180,E1 13557.807,E2 13557.807} C_VEL
LIN {X 0,Y 496.459,Z 901.189,A -85,B 0,C 180,E1 13561.702,E2 13561.702} C_VEL
LIN {X 0,Y 491.865,Z 931.76,A -85,B 0,C 180,E1 13566.093,E2 13566.093} C_VEL
LIN {X 0,Y 490.028,Z 936.81,A -85,B 0,C 180,E1 13566.899,E2 13566.899} C_VEL
LIN {X 0,Y 481.864,Z 949.392,A -85,B 0,C 180,E1 13569.149,E2 13569.149} C_VEL
LIN {X 0,Y 481.636,Z 950.464,A -85,B 0,C 180,E1 13569.375,E2 13569.375} C_VEL
LIN {X 0,Y 479.461,Z 970.837,A -85,B 0,C 180,E1 13574.271,E2 13574.271} C_VEL
LIN {X 0,Y 478.517,Z 985.003,A -85,B 0,C 180,E1 13579.053,E2 13579.053} C_VEL
LIN {X 0,Y 478.246,Z 993.791,A -85,B 0,C 180,E1 13583.638,E2 13583.638} C_VEL
LIN {X 0,Y 478.299,Z 998.024,A -85,B 0,C 180,E1 13588.19,E2 13588.19} C_VEL
LIN {X 0,Y 478.177,Z 998.195,A -85,B 0,C 180,E1 13591.821,E2 13591.821} C_VEL
LIN {X 0,Y 478.193,Z 994.338,A -85,B 0,C 180,E1 13596.372,E2 13596.372} C_VEL
LIN {X 0,Y 478.505,Z 985.817,A -85,B 0,C 180,E1 13601.051,E2 13601.051} C_VEL
LIN {X 0,Y 479.477,Z 972.358,A -85,B 0,C 180,E1 13605.739,E2 13605.739} C_VEL
LIN {X 0,Y 481.794,Z 952.139,A -85,B 0,C 180,E1 13610.725,E2 13610.725} C_VEL
LIN {X 0,Y 485.52,Z 926.148,A -85,B 0,C 180,E1 13615.46,E2 13615.46} C_VEL
LIN {X 0,Y 491.193,Z 892.917,A -85,B 0,C 180,E1 13619.998,E2 13619.998} C_VEL
LIN {X 0,Y 497.435,Z 856.189,A -85,B 0,C 180,E1 13623.775,E2 13623.775} C_VEL
LIN {X 0,Y 504.053,Z 814.66,A -85,B 0,C 180,E1 13626.962,E2 13626.962} C_VEL
LIN {X 0,Y 509.839,Z 772.064,A -85,B 0,C 180,E1 13629.338,E2 13629.338} C_VEL
LIN {X 0,Y 514.8,Z 725.372,A -85,B 0,C 180,E1 13631.104,E2 13631.104} C_VEL
LIN {X 0,Y 516.68,Z 690.443,A -85,B 0,C 180,E1 13631.979,E2 13631.979} C_VEL
LIN {X 0,Y 477.898,Z 606.192,A -85,B 0,C 180,E1 13636.481,E2 13636.481} C_VEL
LIN {X 0,Y 476.172,Z 601.31,A -85,B 0,C 180,E1 13636.744,E2 13636.744} C_VEL
LIN {X 0,Y 476.094,Z 601.31,A -85,B 0,C 180,E1 13642.8,E2 13642.8} C_VEL
LIN {X 0,Y 476.304,Z 601.31,A -85,B 0,C 180,E1 13649.408,E2 13649.408} C_VEL
LIN {X 0,Y 476.554,Z 601.31,A -85,B 0,C 180,E1 13655.589,E2 13655.589} C_VEL
LIN {X 0,Y 476.755,Z 601.31,A -85,B 0,C 180,E1 13661.471,E2 13661.471} C_VEL
LIN {X 0,Y 476.958,Z 601.31,A -85,B 0,C 180,E1 13667.152,E2 13667.152} C_VEL
LIN {X 0,Y 477.274,Z 601.31,A -85,B 0,C 180,E1 13672.704,E2 13672.704} C_VEL
LIN {X 0,Y 477.554,Z 601.31,A -85,B 0,C 180,E1 13678.18,E2 13678.18} C_VEL
LIN {X 0,Y 477.52,Z 601.31,A -85,B 0,C 180,E1 13683.635,E2 13683.635} C_VEL
LIN {X 0,Y 477.089,Z 601.31,A -85,B 0,C 180,E1 13690.059,E2 13690.059} C_VEL
LIN {X 0,Y 476.852,Z 601.31,A -85,B 0,C 180,E1 13696.611,E2 13696.611} C_VEL
LIN {X 0,Y 476.599,Z 601.31,A -85,B 0,C 180,E1 13702.771,E2 13702.771} C_VEL
LIN {X 0,Y 476.399,Z 601.31,A -85,B 0,C 180,E1 13708.486,E2 13708.486} C_VEL
LIN {X 0,Y 476.215,Z 601.31,A -85,B 0,C 180,E1 13714.929,E2 13714.929} C_VEL
LIN {X 0,Y 476.114,Z 601.31,A -85,B 0,C 180,E1 13721.923,E2 13721.923} C_VEL
LIN {X 0,Y 476.082,Z 601.31,A -85,B 0,C 180,E1 13728.053,E2 13728.053} C_VEL
LIN {X 0,Y 476.21,Z 602.064,A -85,B 0,C 180,E1 13732.55,E2 13732.55} C_VEL
LIN {X 0,Y 497.653,Z 649.897,A -85,B 0,C 180,E1 13735.897,E2 13735.897} C_VEL
LIN {X 0,Y 504.762,Z 674.099,A -85,B 0,C 180,E1 13737.369,E2 13737.369} C_VEL
LIN {X 0,Y 501.289,Z 713.745,A -85,B 0,C 180,E1 13739.278,E2 13739.278} C_VEL
LIN {X 0,Y 496.751,Z 749.736,A -85,B 0,C 180,E1 13741.776,E2 13741.776} C_VEL
LIN {X 0,Y 491.825,Z 782.999,A -85,B 0,C 180,E1 13744.932,E2 13744.932} C_VEL
LIN {X 0,Y 487.179,Z 811.854,A -85,B 0,C 180,E1 13748.661,E2 13748.661} C_VEL
LIN {X 0,Y 483.581,Z 835.044,A -85,B 0,C 180,E1 13752.707,E2 13752.707} C_VEL
LIN {X 0,Y 481.04,Z 853.681,A -85,B 0,C 180,E1 13757.257,E2 13757.257} C_VEL
LIN {X 0,Y 479.669,Z 866.033,A -85,B 0,C 180,E1 13761.823,E2 13761.823} C_VEL
LIN {X 0,Y 479.068,Z 872.812,A -85,B 0,C 180,E1 13766.368,E2 13766.368} C_VEL
LIN {X 0,Y 479.04,Z 874.497,A -85,B 0,C 180,E1 13769.995,E2 13769.995} C_VEL
LIN {X 0,Y 479.2,Z 871.948,A -85,B 0,C 180,E1 13774.432,E2 13774.432} C_VEL
LIN {X 0,Y 479.884,Z 863.84,A -85,B 0,C 180,E1 13779.078,E2 13779.078} C_VEL
LIN {X 0,Y 481.512,Z 850.133,A -85,B 0,C 180,E1 13783.646,E2 13783.646} C_VEL
LIN {X 0,Y 484.184,Z 831.057,A -85,B 0,C 180,E1 13787.99,E2 13787.99} C_VEL
LIN {X 0,Y 488.131,Z 805.93,A -85,B 0,C 180,E1 13792.104,E2 13792.104} C_VEL
LIN {X 0,Y 492.696,Z 776.927,A -85,B 0,C 180,E1 13795.619,E2 13795.619} C_VEL
LIN {X 0,Y 497.664,Z 742.859,A -85,B 0,C 180,E1 13798.673,E2 13798.673} C_VEL
LIN {X 0,Y 502.018,Z 706.281,A -85,B 0,C 180,E1 13801.04,E2 13801.04} C_VEL
LIN {X 0,Y 504.445,Z 673.664,A -85,B 0,C 180,E1 13802.574,E2 13802.574} C_VEL
LIN {X 0,Y 497.824,Z 650.558,A -85,B 0,C 180,E1 13803.966,E2 13803.966} C_VEL
LIN {X 0,Y 479.835,Z 610.06,A -85,B 0,C 180,E1 13806.755,E2 13806.755} C_VEL
LIN {X 0,Y 476.275,Z 601.31,A -85,B 0,C 180,E1 13807.396,E2 13807.396} C_VEL
LIN {X 0,Y 476.1,Z 601.31,A -85,B 0,C 180,E1 13814.433,E2 13814.433} C_VEL
LIN {X 0,Y 476.075,Z 601.31,A -85,B 0,C 180,E1 13820.479,E2 13820.479} C_VEL
LIN {X 0,Y 476.213,Z 601.31,A -85,B 0,C 180,E1 13827.265,E2 13827.265} C_VEL
LIN {X 0,Y 476.572,Z 601.334,A -85,B 0,C 180,E1 13832.53,E2 13832.53} C_VEL
LIN {X 0,Y 495.153,Z 659.287,A -85,B 0,C 180,E1 13834.741,E2 13834.741} C_VEL
LIN {X 0,Y 493.139,Z 704.446,A -85,B 0,C 180,E1 13835.814,E2 13835.814} C_VEL
LIN {X 0,Y 490.522,Z 743.218,A -85,B 0,C 180,E1 13837.474,E2 13837.474} C_VEL
LIN {X 0,Y 487.496,Z 778.904,A -85,B 0,C 180,E1 13839.783,E2 13839.783} C_VEL
LIN {X 0,Y 484.699,Z 810.155,A -85,B 0,C 180,E1 13842.644,E2 13842.644} C_VEL
LIN {X 0,Y 482.317,Z 836.416,A -85,B 0,C 180,E1 13845.961,E2 13845.961} C_VEL
LIN {X 0,Y 480.78,Z 856.885,A -85,B 0,C 180,E1 13849.564,E2 13849.564} C_VEL
LIN {X 0,Y 479.943,Z 871.204,A -85,B 0,C 180,E1 13853.225,E2 13853.225} C_VEL
LIN {X 0,Y 479.71,Z 880.789,A -85,B 0,C 180,E1 13857.287,E2 13857.287} C_VEL
LIN {X 0,Y 479.715,Z 883.779,A -85,B 0,C 180,E1 13860.002,E2 13860.002} C_VEL
LIN {X 0,Y 480.175,Z 883.569,A -85,B 0,C 180,E1 13863.62,E2 13863.62} C_VEL
LIN {X 0,Y 481.303,Z 878.448,A -85,B 0,C 180,E1 13867.235,E2 13867.235} C_VEL
LIN {X 0,Y 483.119,Z 867.96,A -85,B 0,C 180,E1 13870.846,E2 13870.846} C_VEL
LIN {X 0,Y 485.574,Z 851.392,A -85,B 0,C 180,E1 13874.455,E2 13874.455} C_VEL
LIN {X 0,Y 488.942,Z 828.929,A -85,B 0,C 180,E1 13877.818,E2 13877.818} C_VEL
LIN {X 0,Y 493.025,Z 799.878,A -85,B 0,C 180,E1 13880.93,E2 13880.93} C_VEL
LIN {X 0,Y 497.571,Z 765.403,A -85,B 0,C 180,E1 13883.578,E2 13883.578} C_VEL
LIN {X 0,Y 502.524,Z 725.852,A -85,B 0,C 180,E1 13885.742,E2 13885.742} C_VEL
LIN {X 0,Y 507.615,Z 681.57,A -85,B 0,C 180,E1 13887.349,E2 13887.349} C_VEL
LIN {X 0,Y 508.75,Z 665.468,A -85,B 0,C 180,E1 13887.86,E2 13887.86} C_VEL
LIN {X 0,Y 501.664,Z 644.702,A -85,B 0,C 180,E1 13889.795,E2 13889.795} C_VEL
LIN {X 0,Y 494.054,Z 628.495,A -85,B 0,C 180,E1 13892.288,E2 13892.288} C_VEL
LIN {X 0,Y 490.192,Z 622.196,A -85,B 0,C 180,E1 13894.035,E2 13894.035} C_VEL
LIN {X 0,Y 487.717,Z 616.493,A -85,B 0,C 180,E1 13896.633,E2 13896.633} C_VEL
LIN {X 0,Y 488.132,Z 617.489,A -85,B 0,C 180,E1 13898.857,E2 13898.857} C_VEL
LIN {X 0,Y 492.332,Z 624.695,A -85,B 0,C 180,E1 13901.536,E2 13901.536} C_VEL
LIN {X 0,Y 498.595,Z 635.306,A -85,B 0,C 180,E1 13903.614,E2 13903.614} C_VEL
LIN {X 0,Y 506.492,Z 651.648,A -85,B 0,C 180,E1 13905.528,E2 13905.528} C_VEL
LIN {X 0,Y 513.642,Z 672.876,A -85,B 0,C 180,E1 13907.037,E2 13907.037} C_VEL
LIN {X 0,Y 517.913,Z 693.71,A -85,B 0,C 180,E1 13908.052,E2 13908.052} C_VEL
LIN {X 0,Y 513.435,Z 740.353,A -85,B 0,C 180,E1 13909.386,E2 13909.386} C_VEL
LIN {X 0,Y 507.714,Z 784.85,A -85,B 0,C 180,E1 13911.395,E2 13911.395} C_VEL
LIN {X 0,Y 501.494,Z 826.333,A -85,B 0,C 180,E1 13914.042,E2 13914.042} C_VEL
LIN {X 0,Y 495.073,Z 865.117,A -85,B 0,C 180,E1 13917.348,E2 13917.348} C_VEL
LIN {X 0,Y 489.05,Z 900.507,A -85,B 0,C 180,E1 13921.305,E2 13921.305} C_VEL
LIN {X 0,Y 484.034,Z 932.371,A -85,B 0,C 180,E1 13925.992,E2 13925.992} C_VEL
LIN {X 0,Y 481.636,Z 950.464,A -85,B 0,C 180,E1 13929.375,E2 13929.375} C_VEL
LIN {X 0,Y 476.694,Z 958.666,A -85,B 0,C 180,E1 13931.136,E2 13931.136} C_VEL
LIN {X 0,Y 471.98,Z 966.081,A -85,B 0,C 180,E1 13932.972,E2 13932.972} C_VEL
LIN {X 0,Y 470.77,Z 981.755,A -85,B 0,C 180,E1 13937.929,E2 13937.929} C_VEL
LIN {X 0,Y 470.426,Z 991.479,A -85,B 0,C 180,E1 13942.603,E2 13942.603} C_VEL
LIN {X 0,Y 470.373,Z 996.286,A -85,B 0,C 180,E1 13946.785,E2 13946.785} C_VEL
LIN {X 0,Y 470.517,Z 997.594,A -85,B 0,C 180,E1 13950.005,E2 13950.005} C_VEL
LIN {X 0,Y 470.419,Z 996.316,A -85,B 0,C 180,E1 13953.699,E2 13953.699} C_VEL
LIN {X 0,Y 470.319,Z 990.618,A -85,B 0,C 180,E1 13958.341,E2 13958.341} C_VEL
LIN {X 0,Y 471.009,Z 979.107,A -85,B 0,C 180,E1 13963.492,E2 13963.492} C_VEL
LIN {X 0,Y 472.662,Z 961.237,A -85,B 0,C 180,E1 13968.703,E2 13968.703} C_VEL
LIN {X 0,Y 475.821,Z 938.711,A -85,B 0,C 180,E1 13973.462,E2 13973.462} C_VEL
LIN {X 0,Y 480.473,Z 910.791,A -85,B 0,C 180,E1 13977.934,E2 13977.934} C_VEL
LIN {X 0,Y 486.085,Z 878.94,A -85,B 0,C 180,E1 13981.85,E2 13981.85} C_VEL
LIN {X 0,Y 492.444,Z 842.4,A -85,B 0,C 180,E1 13985.291,E2 13985.291} C_VEL
LIN {X 0,Y 498.858,Z 801.777,A -85,B 0,C 180,E1 13988.154,E2 13988.154} C_VEL
LIN {X 0,Y 504.718,Z 757.551,A -85,B 0,C 180,E1 13990.39,E2 13990.39} C_VEL
LIN {X 0,Y 509.22,Z 709.691,A -85,B 0,C 180,E1 13991.977,E2 13991.977} C_VEL
LIN {X 0,Y 509.691,Z 692.445,A -85,B 0,C 180,E1 13992.402,E2 13992.402} C_VEL
LIN {X 0,Y 471.701,Z 610.167,A -85,B 0,C 180,E1 13996.878,E2 13996.878} C_VEL
LIN {X 0,Y 468.212,Z 601.31,A -85,B 0,C 180,E1 13997.444,E2 13997.444} C_VEL
LIN {X 0,Y 468.163,Z 601.31,A -85,B 0,C 180,E1 14004.375,E2 14004.375} C_VEL
LIN {X 0,Y 468.332,Z 601.31,A -85,B 0,C 180,E1 14008.83,E2 14008.83} C_VEL
LIN {X 0,Y 468.579,Z 601.31,A -85,B 0,C 180,E1 14015.145,E2 14015.145} C_VEL
LIN {X 0,Y 468.809,Z 601.31,A -85,B 0,C 180,E1 14021.145,E2 14021.145} C_VEL
LIN {X 0,Y 469.021,Z 601.31,A -85,B 0,C 180,E1 14026.931,E2 14026.931} C_VEL
LIN {X 0,Y 469.354,Z 601.31,A -85,B 0,C 180,E1 14032.58,E2 14032.58} C_VEL
LIN {X 0,Y 469.657,Z 601.31,A -85,B 0,C 180,E1 14038.149,E2 14038.149} C_VEL
LIN {X 0,Y 469.609,Z 601.31,A -85,B 0,C 180,E1 14043.697,E2 14043.697} C_VEL
LIN {X 0,Y 469.256,Z 601.31,A -85,B 0,C 180,E1 14049.287,E2 14049.287} C_VEL
LIN {X 0,Y 469.006,Z 601.31,A -85,B 0,C 180,E1 14054.973,E2 14054.973} C_VEL
LIN {X 0,Y 468.778,Z 601.31,A -85,B 0,C 180,E1 14060.82,E2 14060.82} C_VEL
LIN {X 0,Y 468.496,Z 601.31,A -85,B 0,C 180,E1 14066.914,E2 14066.914} C_VEL
LIN {X 0,Y 468.302,Z 601.31,A -85,B 0,C 180,E1 14073.359,E2 14073.359} C_VEL
LIN {X 0,Y 468.218,Z 601.31,A -85,B 0,C 180,E1 14080.319,E2 14080.319} C_VEL
LIN {X 0,Y 468.213,Z 601.31,A -85,B 0,C 180,E1 14085.378,E2 14085.378} C_VEL
LIN {X 0,Y 468.305,Z 601.762,A -85,B 0,C 180,E1 14091.761,E2 14091.761} C_VEL
LIN {X 0,Y 490.734,Z 651.572,A -85,B 0,C 180,E1 14095.391,E2 14095.391} C_VEL
LIN {X 0,Y 498.157,Z 676.863,A -85,B 0,C 180,E1 14096.979,E2 14096.979} C_VEL
LIN {X 0,Y 494.469,Z 715.32,A -85,B 0,C 180,E1 14098.86,E2 14098.86} C_VEL
LIN {X 0,Y 489.843,Z 750.647,A -85,B 0,C 180,E1 14101.345,E2 14101.345} C_VEL
LIN {X 0,Y 484.87,Z 782.96,A -85,B 0,C 180,E1 14104.437,E2 14104.437} C_VEL
LIN {X 0,Y 479.971,Z 811.986,A -85,B 0,C 180,E1 14108.191,E2 14108.191} C_VEL
LIN {X 0,Y 476.146,Z 835.548,A -85,B 0,C 180,E1 14112.333,E2 14112.333} C_VEL
LIN {X 0,Y 473.577,Z 853.092,A -85,B 0,C 180,E1 14116.582,E2 14116.582} C_VEL
LIN {X 0,Y 472.105,Z 865.029,A -85,B 0,C 180,E1 14120.76,E2 14120.76} C_VEL
LIN {X 0,Y 471.37,Z 872.454,A -85,B 0,C 180,E1 14125.024,E2 14125.024} C_VEL
LIN {X 0,Y 471.218,Z 875.483,A -85,B 0,C 180,E1 14129.995,E2 14129.995} C_VEL
LIN {X 0,Y 471.394,Z 872.29,A -85,B 0,C 180,E1 14135.009,E2 14135.009} C_VEL
LIN {X 0,Y 472.117,Z 864.822,A -85,B 0,C 180,E1 14139.229,E2 14139.229} C_VEL
LIN {X 0,Y 473.85,Z 851.114,A -85,B 0,C 180,E1 14143.871,E2 14143.871} C_VEL
LIN {X 0,Y 476.544,Z 832.771,A -85,B 0,C 180,E1 14148.134,E2 14148.134} C_VEL
LIN {X 0,Y 480.56,Z 808.517,A -85,B 0,C 180,E1 14152.227,E2 14152.227} C_VEL
LIN {X 0,Y 485.192,Z 780.501,A -85,B 0,C 180,E1 14155.735,E2 14155.735} C_VEL
LIN {X 0,Y 490.36,Z 746.941,A -85,B 0,C 180,E1 14158.864,E2 14158.864} C_VEL
LIN {X 0,Y 494.825,Z 711.639,A -85,B 0,C 180,E1 14161.252,E2 14161.252} C_VEL
LIN {X 0,Y 497.603,Z 675.293,A -85,B 0,C 180,E1 14163.035,E2 14163.035} C_VEL
LIN {X 0,Y 490.737,Z 651.98,A -85,B 0,C 180,E1 14164.494,E2 14164.494} C_VEL
LIN {X 0,Y 472.776,Z 611.458,A -85,B 0,C 180,E1 14167.378,E2 14167.378} C_VEL
LIN {X 0,Y 468.368,Z 601.31,A -85,B 0,C 180,E1 14168.173,E2 14168.173} C_VEL
LIN {X 0,Y 468.212,Z 601.31,A -85,B 0,C 180,E1 14174.622,E2 14174.622} C_VEL
LIN {X 0,Y 468.135,Z 601.31,A -85,B 0,C 180,E1 14180.961,E2 14180.961} C_VEL
LIN {X 0,Y 468.335,Z 601.31,A -85,B 0,C 180,E1 14187.255,E2 14187.255} C_VEL
LIN {X 0,Y 468.647,Z 602.032,A -85,B 0,C 180,E1 14192.102,E2 14192.102} C_VEL
LIN {X 0,Y 487.76,Z 660.734,A -85,B 0,C 180,E1 14194.421,E2 14194.421} C_VEL
LIN {X 0,Y 485.644,Z 705.963,A -85,B 0,C 180,E1 14195.541,E2 14195.541} C_VEL
LIN {X 0,Y 482.977,Z 744.289,A -85,B 0,C 180,E1 14197.224,E2 14197.224} C_VEL
LIN {X 0,Y 479.846,Z 779.963,A -85,B 0,C 180,E1 14199.577,E2 14199.577} C_VEL
LIN {X 0,Y 476.995,Z 811.138,A -85,B 0,C 180,E1 14202.481,E2 14202.481} C_VEL
LIN {X 0,Y 474.499,Z 837.825,A -85,B 0,C 180,E1 14205.913,E2 14205.913} C_VEL
LIN {X 0,Y 472.921,Z 858.409,A -85,B 0,C 180,E1 14209.622,E2 14209.622} C_VEL
LIN {X 0,Y 472.041,Z 873.556,A -85,B 0,C 180,E1 14213.646,E2 14213.646} C_VEL
LIN {X 0,Y 471.901,Z 881.695,A -85,B 0,C 180,E1 14217.242,E2 14217.242} C_VEL
LIN {X 0,Y 471.894,Z 884.811,A -85,B 0,C 180,E1 14220.002,E2 14220.002} C_VEL
LIN {X 0,Y 472.402,Z 884.78,A -85,B 0,C 180,E1 14223.68,E2 14223.68} C_VEL
LIN {X 0,Y 473.616,Z 879.709,A -85,B 0,C 180,E1 14227.4,E2 14227.4} C_VEL
LIN {X 0,Y 475.519,Z 869.546,A -85,B 0,C 180,E1 14231.022,E2 14231.022} C_VEL
LIN {X 0,Y 478.134,Z 853.192,A -85,B 0,C 180,E1 14234.685,E2 14234.685} C_VEL
LIN {X 0,Y 481.731,Z 831.104,A -85,B 0,C 180,E1 14238.094,E2 14238.094} C_VEL
LIN {X 0,Y 486.023,Z 802.563,A -85,B 0,C 180,E1 14241.246,E2 14241.246} C_VEL
LIN {X 0,Y 490.985,Z 768.037,A -85,B 0,C 180,E1 14244.002,E2 14244.002} C_VEL
LIN {X 0,Y 496.381,Z 728.092,A -85,B 0,C 180,E1 14246.267,E2 14246.267} C_VEL
LIN {X 0,Y 501.938,Z 684.195,A -85,B 0,C 180,E1 14247.939,E2 14247.939} C_VEL
LIN {X 0,Y 503.199,Z 667.872,A -85,B 0,C 180,E1 14248.486,E2 14248.486} C_VEL
LIN {X 0,Y 496.651,Z 648.145,A -85,B 0,C 180,E1 14250.489,E2 14250.489} C_VEL
LIN {X 0,Y 490.702,Z 635.036,A -85,B 0,C 180,E1 14252.693,E2 14252.693} C_VEL
LIN {X 0,Y 487.444,Z 629.233,A -85,B 0,C 180,E1 14254.406,E2 14254.406} C_VEL
LIN {X 0,Y 485.876,Z 624.639,A -85,B 0,C 180,E1 14256.329,E2 14256.329} C_VEL
LIN {X 0,Y 486.219,Z 625.5,A -85,B 0,C 180,E1 14258.832,E2 14258.832} C_VEL
LIN {X 0,Y 489.998,Z 632.228,A -85,B 0,C 180,E1 14261.331,E2 14261.331} C_VEL
LIN {X 0,Y 495.805,Z 642.63,A -85,B 0,C 180,E1 14263.367,E2 14263.367} C_VEL
LIN {X 0,Y 503.079,Z 658.966,A -85,B 0,C 180,E1 14265.246,E2 14265.246} C_VEL
LIN {X 0,Y 509.177,Z 679.553,A -85,B 0,C 180,E1 14266.673,E2 14266.673} C_VEL
LIN {X 0,Y 512.05,Z 695.939,A -85,B 0,C 180,E1 14267.491,E2 14267.491} C_VEL
LIN {X 0,Y 507.243,Z 741.703,A -85,B 0,C 180,E1 14268.857,E2 14268.857} C_VEL
LIN {X 0,Y 501.23,Z 785.288,A -85,B 0,C 180,E1 14270.879,E2 14270.879} C_VEL
LIN {X 0,Y 494.598,Z 826.869,A -85,B 0,C 180,E1 14273.596,E2 14273.596} C_VEL
LIN {X 0,Y 487.81,Z 865.626,A -85,B 0,C 180,E1 14276.984,E2 14276.984} C_VEL
LIN {X 0,Y 481.8,Z 899.404,A -85,B 0,C 180,E1 14280.832,E2 14280.832} C_VEL
LIN {X 0,Y 476.452,Z 931.275,A -85,B 0,C 180,E1 14285.585,E2 14285.585} C_VEL
LIN {X 0,Y 472.907,Z 956.942,A -85,B 0,C 180,E1 14290.682,E2 14290.682} C_VEL
LIN {X 0,Y 471.98,Z 966.081,A -85,B 0,C 180,E1 14292.972,E2 14292.972} C_VEL
LIN {X 0,Y 469.031,Z 971.199,A -85,B 0,C 180,E1 14294.406,E2 14294.406} C_VEL
LIN {X 0,Y 463.183,Z 977.74,A -85,B 0,C 180,E1 14296.594,E2 14296.594} C_VEL
LIN {X 0,Y 463.051,Z 978.435,A -85,B 0,C 180,E1 14296.852,E2 14296.852} C_VEL
LIN {X 0,Y 462.592,Z 989.005,A -85,B 0,C 180,E1 14301.529,E2 14301.529} C_VEL
LIN {X 0,Y 462.52,Z 995.052,A -85,B 0,C 180,E1 14306.249,E2 14306.249} C_VEL
LIN {X 0,Y 462.667,Z 996.688,A -85,B 0,C 180,E1 14310.005,E2 14310.005} C_VEL
LIN {X 0,Y 462.565,Z 995.409,A -85,B 0,C 180,E1 14313.762,E2 14313.762} C_VEL
LIN {X 0,Y 462.476,Z 989.647,A -85,B 0,C 180,E1 14318.483,E2 14318.483} C_VEL
LIN {X 0,Y 463.138,Z 978.038,A -85,B 0,C 180,E1 14323.726,E2 14323.726} C_VEL
LIN {X 0,Y 464.906,Z 959.76,A -85,B 0,C 180,E1 14329.092,E2 14329.092} C_VEL
LIN {X 0,Y 468.471,Z 935.989,A -85,B 0,C 180,E1 14334.106,E2 14334.106} C_VEL
LIN {X 0,Y 473.44,Z 906.986,A -85,B 0,C 180,E1 14338.695,E2 14338.695} C_VEL
LIN {X 0,Y 479.168,Z 875.424,A -85,B 0,C 180,E1 14342.524,E2 14342.524} C_VEL
LIN {X 0,Y 485.558,Z 839.694,A -85,B 0,C 180,E1 14345.861,E2 14345.861} C_VEL
LIN {X 0,Y 492.153,Z 798.954,A -85,B 0,C 180,E1 14348.715,E2 14348.715} C_VEL
LIN {X 0,Y 497.908,Z 756.207,A -85,B 0,C 180,E1 14350.869,E2 14350.869} C_VEL
LIN {X 0,Y 502.317,Z 710.581,A -85,B 0,C 180,E1 14352.403,E2 14352.403} C_VEL
LIN {X 0,Y 502.731,Z 694.601,A -85,B 0,C 180,E1 14352.82,E2 14352.82} C_VEL
LIN {X 0,Y 465.248,Z 613.331,A -85,B 0,C 180,E1 14357.326,E2 14357.326} C_VEL
LIN {X 0,Y 460.295,Z 601.31,A -85,B 0,C 180,E1 14358.036,E2 14358.036} C_VEL
LIN {X 0,Y 460.234,Z 601.31,A -85,B 0,C 180,E1 14363.664,E2 14363.664} C_VEL
LIN {X 0,Y 460.463,Z 601.31,A -85,B 0,C 180,E1 14370.427,E2 14370.427} C_VEL
LIN {X 0,Y 460.803,Z 601.31,A -85,B 0,C 180,E1 14377.041,E2 14377.041} C_VEL
LIN {X 0,Y 460.943,Z 601.31,A -85,B 0,C 180,E1 14382.793,E2 14382.793} C_VEL
LIN {X 0,Y 461.194,Z 601.31,A -85,B 0,C 180,E1 14388.631,E2 14388.631} C_VEL
LIN {X 0,Y 461.583,Z 601.31,A -85,B 0,C 180,E1 14394.347,E2 14394.347} C_VEL
LIN {X 0,Y 461.903,Z 601.31,A -85,B 0,C 180,E1 14399.998,E2 14399.998} C_VEL
LIN {X 0,Y 461.596,Z 601.31,A -85,B 0,C 180,E1 14405.648,E2 14405.648} C_VEL
LIN {X 0,Y 461.238,Z 601.31,A -85,B 0,C 180,E1 14411.363,E2 14411.363} C_VEL
LIN {X 0,Y 460.929,Z 601.31,A -85,B 0,C 180,E1 14417.56,E2 14417.56} C_VEL
LIN {X 0,Y 460.753,Z 601.31,A -85,B 0,C 180,E1 14423.235,E2 14423.235} C_VEL
LIN {X 0,Y 460.455,Z 601.31,A -85,B 0,C 180,E1 14429.568,E2 14429.568} C_VEL
LIN {X 0,Y 460.29,Z 601.31,A -85,B 0,C 180,E1 14436.325,E2 14436.325} C_VEL
LIN {X 0,Y 460.293,Z 601.31,A -85,B 0,C 180,E1 14441.162,E2 14441.162} C_VEL
LIN {X 0,Y 460.252,Z 601.31,A -85,B 0,C 180,E1 14446.392,E2 14446.392} C_VEL
LIN {X 0,Y 460.3,Z 601.503,A -85,B 0,C 180,E1 14450.923,E2 14450.923} C_VEL
LIN {X 0,Y 483.275,Z 651.842,A -85,B 0,C 180,E1 14454.769,E2 14454.769} C_VEL
LIN {X 0,Y 491.427,Z 678.533,A -85,B 0,C 180,E1 14456.516,E2 14456.516} C_VEL
LIN {X 0,Y 487.479,Z 718.228,A -85,B 0,C 180,E1 14458.511,E2 14458.511} C_VEL
LIN {X 0,Y 482.564,Z 753.998,A -85,B 0,C 180,E1 14461.102,E2 14461.102} C_VEL
LIN {X 0,Y 477.18,Z 787.21,A -85,B 0,C 180,E1 14464.405,E2 14464.405} C_VEL
LIN {X 0,Y 472.283,Z 815.17,A -85,B 0,C 180,E1 14468.185,E2 14468.185} C_VEL
LIN {X 0,Y 468.269,Z 838.739,A -85,B 0,C 180,E1 14472.5,E2 14472.5} C_VEL
LIN {X 0,Y 465.68,Z 855.647,A -85,B 0,C 180,E1 14476.829,E2 14476.829} C_VEL
LIN {X 0,Y 464.125,Z 868.001,A -85,B 0,C 180,E1 14481.547,E2 14481.547} C_VEL
LIN {X 0,Y 463.421,Z 874.785,A -85,B 0,C 180,E1 14486.245,E2 14486.245} C_VEL
LIN {X 0,Y 463.391,Z 876.47,A -85,B 0,C 180,E1 14489.995,E2 14489.995} C_VEL
LIN {X 0,Y 463.531,Z 873.926,A -85,B 0,C 180,E1 14494.579,E2 14494.579} C_VEL
LIN {X 0,Y 464.344,Z 865.808,A -85,B 0,C 180,E1 14499.385,E2 14499.385} C_VEL
LIN {X 0,Y 466.214,Z 852.096,A -85,B 0,C 180,E1 14504.103,E2 14504.103} C_VEL
LIN {X 0,Y 469.119,Z 833.437,A -85,B 0,C 180,E1 14508.498,E2 14508.498} C_VEL
LIN {X 0,Y 473.277,Z 809.466,A -85,B 0,C 180,E1 14512.587,E2 14512.587} C_VEL
LIN {X 0,Y 478.376,Z 779.866,A -85,B 0,C 180,E1 14516.318,E2 14516.318} C_VEL
LIN {X 0,Y 483.69,Z 746.377,A -85,B 0,C 180,E1 14519.428,E2 14519.428} C_VEL
LIN {X 0,Y 488.316,Z 710.688,A -85,B 0,C 180,E1 14521.831,E2 14521.831} C_VEL
LIN {X 0,Y 490.929,Z 677.28,A -85,B 0,C 180,E1 14523.48,E2 14523.48} C_VEL
LIN {X 0,Y 483.883,Z 653.891,A -85,B 0,C 180,E1 14525.004,E2 14525.004} C_VEL
LIN {X 0,Y 466.648,Z 615.192,A -85,B 0,C 180,E1 14527.858,E2 14527.858} C_VEL
LIN {X 0,Y 460.39,Z 601.31,A -85,B 0,C 180,E1 14529.034,E2 14529.034} C_VEL
LIN {X 0,Y 460.273,Z 601.31,A -85,B 0,C 180,E1 14533.727,E2 14533.727} C_VEL
LIN {X 0,Y 460.257,Z 601.31,A -85,B 0,C 180,E1 14539.208,E2 14539.208} C_VEL
LIN {X 0,Y 460.281,Z 601.31,A -85,B 0,C 180,E1 14545.981,E2 14545.981} C_VEL
LIN {X 0,Y 460.668,Z 601.31,A -85,B 0,C 180,E1 14551.606,E2 14551.606} C_VEL
LIN {X 0,Y 480.427,Z 661.69,A -85,B 0,C 180,E1 14554.089,E2 14554.089} C_VEL
LIN {X 0,Y 478.25,Z 706.113,A -85,B 0,C 180,E1 14555.211,E2 14555.211} C_VEL
LIN {X 0,Y 475.462,Z 745.317,A -85,B 0,C 180,E1 14556.967,E2 14556.967} C_VEL
LIN {X 0,Y 472.232,Z 780.707,A -85,B 0,C 180,E1 14559.339,E2 14559.339} C_VEL
LIN {X 0,Y 469.298,Z 812.015,A -85,B 0,C 180,E1 14562.3,E2 14562.3} C_VEL
LIN {X 0,Y 466.794,Z 837.99,A -85,B 0,C 180,E1 14565.676,E2 14565.676} C_VEL
LIN {X 0,Y 465.14,Z 858.868,A -85,B 0,C 180,E1 14569.446,E2 14569.446} C_VEL
LIN {X 0,Y 464.243,Z 873.942,A -85,B 0,C 180,E1 14573.444,E2 14573.444} C_VEL
LIN {X 0,Y 464.059,Z 882.602,A -85,B 0,C 180,E1 14577.196,E2 14577.196} C_VEL
LIN {X 0,Y 464.075,Z 885.844,A -85,B 0,C 180,E1 14580.002,E2 14580.002} C_VEL
LIN {X 0,Y 464.62,Z 885.993,A -85,B 0,C 180,E1 14583.741,E2 14583.741} C_VEL
LIN {X 0,Y 465.89,Z 881.198,A -85,B 0,C 180,E1 14587.476,E2 14587.476} C_VEL
LIN {X 0,Y 467.944,Z 871.157,A -85,B 0,C 180,E1 14591.203,E2 14591.203} C_VEL
LIN {X 0,Y 470.718,Z 855.056,A -85,B 0,C 180,E1 14594.922,E2 14594.922} C_VEL
LIN {X 0,Y 474.547,Z 833.364,A -85,B 0,C 180,E1 14598.377,E2 14598.377} C_VEL
LIN {X 0,Y 479.265,Z 804.256,A -85,B 0,C 180,E1 14601.683,E2 14601.683} C_VEL
LIN {X 0,Y 484.534,Z 770.28,A -85,B 0,C 180,E1 14604.474,E2 14604.474} C_VEL
LIN {X 0,Y 490.531,Z 729.774,A -85,B 0,C 180,E1 14606.852,E2 14606.852} C_VEL
LIN {X 0,Y 496.574,Z 686.424,A -85,B 0,C 180,E1 14608.565,E2 14608.565} C_VEL
LIN {X 0,Y 497.997,Z 670.838,A -85,B 0,C 180,E1 14609.102,E2 14609.102} C_VEL
LIN {X 0,Y 492.179,Z 652.541,A -85,B 0,C 180,E1 14611.119,E2 14611.119} C_VEL
LIN {X 0,Y 487.244,Z 641.088,A -85,B 0,C 180,E1 14613.242,E2 14613.242} C_VEL
LIN {X 0,Y 484.879,Z 636.303,A -85,B 0,C 180,E1 14614.748,E2 14614.748} C_VEL
LIN {X 0,Y 483.835,Z 632.249,A -85,B 0,C 180,E1 14616.507,E2 14616.507} C_VEL
LIN {X 0,Y 484.268,Z 633.254,A -85,B 0,C 180,E1 14618.732,E2 14618.732} C_VEL
LIN {X 0,Y 487.691,Z 639.714,A -85,B 0,C 180,E1 14621.12,E2 14621.12} C_VEL
LIN {X 0,Y 493.647,Z 651.039,A -85,B 0,C 180,E1 14623.292,E2 14623.292} C_VEL
LIN {X 0,Y 500.327,Z 668.499,A -85,B 0,C 180,E1 14625.128,E2 14625.128} C_VEL
LIN {X 0,Y 505.562,Z 690.958,A -85,B 0,C 180,E1 14626.552,E2 14626.552} C_VEL
LIN {X 0,Y 506.321,Z 698.56,A -85,B 0,C 180,E1 14626.915,E2 14626.915} C_VEL
LIN {X 0,Y 501.162,Z 743.278,A -85,B 0,C 180,E1 14628.313,E2 14628.313} C_VEL
LIN {X 0,Y 494.692,Z 786.84,A -85,B 0,C 180,E1 14630.403,E2 14630.403} C_VEL
LIN {X 0,Y 487.735,Z 827.688,A -85,B 0,C 180,E1 14633.15,E2 14633.15} C_VEL
LIN {X 0,Y 480.918,Z 864.673,A -85,B 0,C 180,E1 14636.449,E2 14636.449} C_VEL
LIN {X 0,Y 474.215,Z 900.127,A -85,B 0,C 180,E1 14640.582,E2 14640.582} C_VEL
LIN {X 0,Y 468.948,Z 930.232,A -85,B 0,C 180,E1 14645.169,E2 14645.169} C_VEL
LIN {X 0,Y 465.266,Z 955.533,A -85,B 0,C 180,E1 14650.259,E2 14650.259} C_VEL
LIN {X 0,Y 463.347,Z 974.001,A -85,B 0,C 180,E1 14655.324,E2 14655.324} C_VEL
LIN {X 0,Y 463.051,Z 978.435,A -85,B 0,C 180,E1 14656.852,E2 14656.852} C_VEL
LIN {X 0,Y 460.33,Z 982.268,A -85,B 0,C 180,E1 14658.377,E2 14658.377} C_VEL
LIN {X 0,Y 454.816,Z 986.822,A -85,B 0,C 180,E1 14660.7,E2 14660.7} C_VEL
LIN {X 0,Y 454.714,Z 987.314,A -85,B 0,C 180,E1 14660.97,E2 14660.97} C_VEL
LIN {X 0,Y 454.729,Z 992.263,A -85,B 0,C 180,E1 14664.268,E2 14664.268} C_VEL
LIN {X 0,Y 454.757,Z 995.323,A -85,B 0,C 180,E1 14668.096,E2 14668.096} C_VEL
LIN {X 0,Y 454.637,Z 995.483,A -85,B 0,C 180,E1 14671.915,E2 14671.915} C_VEL
LIN {X 0,Y 454.612,Z 991.51,A -85,B 0,C 180,E1 14676.704,E2 14676.704} C_VEL
LIN {X 0,Y 454.955,Z 981.896,A -85,B 0,C 180,E1 14682.02,E2 14682.02} C_VEL
LIN {X 0,Y 456.263,Z 966.141,A -85,B 0,C 180,E1 14687.396,E2 14687.396} C_VEL
LIN {X 0,Y 459.089,Z 944.928,A -85,B 0,C 180,E1 14692.486,E2 14692.486} C_VEL
LIN {X 0,Y 463.496,Z 919.544,A -85,B 0,C 180,E1 14697.059,E2 14697.059} C_VEL
LIN {X 0,Y 469.126,Z 889.155,A -85,B 0,C 180,E1 14701.258,E2 14701.258} C_VEL
LIN {X 0,Y 475.645,Z 853.861,A -85,B 0,C 180,E1 14704.994,E2 14704.994} C_VEL
LIN {X 0,Y 482.534,Z 814.146,A -85,B 0,C 180,E1 14708.148,E2 14708.148} C_VEL
LIN {X 0,Y 489,Z 770.412,A -85,B 0,C 180,E1 14710.671,E2 14710.671} C_VEL
LIN {X 0,Y 494.154,Z 725.74,A -85,B 0,C 180,E1 14712.428,E2 14712.428} C_VEL
LIN {X 0,Y 495.788,Z 696.822,A -85,B 0,C 180,E1 14713.232,E2 14713.232} C_VEL
LIN {X 0,Y 458.048,Z 614.75,A -85,B 0,C 180,E1 14717.872,E2 14717.872} C_VEL
LIN {X 0,Y 452.342,Z 601.31,A -85,B 0,C 180,E1 14718.765,E2 14718.765} C_VEL
LIN {X 0,Y 452.336,Z 601.31,A -85,B 0,C 180,E1 14725.293,E2 14725.293} C_VEL
LIN {X 0,Y 452.556,Z 601.31,A -85,B 0,C 180,E1 14732.052,E2 14732.052} C_VEL
LIN {X 0,Y 452.885,Z 601.31,A -85,B 0,C 180,E1 14738.408,E2 14738.408} C_VEL
LIN {X 0,Y 453.071,Z 601.31,A -85,B 0,C 180,E1 14744.483,E2 14744.483} C_VEL
LIN {X 0,Y 453.42,Z 601.31,A -85,B 0,C 180,E1 14750.381,E2 14750.381} C_VEL
LIN {X 0,Y 453.788,Z 601.31,A -85,B 0,C 180,E1 14756.169,E2 14756.169} C_VEL
LIN {X 0,Y 453.938,Z 601.31,A -85,B 0,C 180,E1 14761.91,E2 14761.91} C_VEL
LIN {X 0,Y 453.514,Z 601.31,A -85,B 0,C 180,E1 14767.676,E2 14767.676} C_VEL
LIN {X 0,Y 453.152,Z 601.31,A -85,B 0,C 180,E1 14774.125,E2 14774.125} C_VEL
LIN {X 0,Y 452.908,Z 601.31,A -85,B 0,C 180,E1 14780.474,E2 14780.474} C_VEL
LIN {X 0,Y 452.643,Z 601.31,A -85,B 0,C 180,E1 14785.787,E2 14785.787} C_VEL
LIN {X 0,Y 452.414,Z 601.31,A -85,B 0,C 180,E1 14792.392,E2 14792.392} C_VEL
LIN {X 0,Y 452.36,Z 601.31,A -85,B 0,C 180,E1 14797.067,E2 14797.067} C_VEL
LIN {X 0,Y 452.275,Z 601.31,A -85,B 0,C 180,E1 14802.512,E2 14802.512} C_VEL
LIN {X 0,Y 452.35,Z 601.31,A -85,B 0,C 180,E1 14809.392,E2 14809.392} C_VEL
LIN {X 0,Y 452.345,Z 601.31,A -85,B 0,C 180,E1 14810.031,E2 14810.031} C_VEL
LIN {X 0,Y 475.616,Z 651.654,A -85,B 0,C 180,E1 14814.092,E2 14814.092} C_VEL
LIN {X 0,Y 484.595,Z 679.612,A -85,B 0,C 180,E1 14816,E2 14816} C_VEL
LIN {X 0,Y 480.902,Z 718.574,A -85,B 0,C 180,E1 14817.992,E2 14817.992} C_VEL
LIN {X 0,Y 475.874,Z 753.816,A -85,B 0,C 180,E1 14820.553,E2 14820.553} C_VEL
LIN {X 0,Y 470.356,Z 786.898,A -85,B 0,C 180,E1 14823.843,E2 14823.843} C_VEL
LIN {X 0,Y 465.214,Z 814.854,A -85,B 0,C 180,E1 14827.621,E2 14827.621} C_VEL
LIN {X 0,Y 460.995,Z 838.255,A -85,B 0,C 180,E1 14831.899,E2 14831.899} C_VEL
LIN {X 0,Y 458.018,Z 856.634,A -85,B 0,C 180,E1 14836.605,E2 14836.605} C_VEL
LIN {X 0,Y 456.363,Z 868.987,A -85,B 0,C 180,E1 14841.402,E2 14841.402} C_VEL
LIN {X 0,Y 455.602,Z 875.772,A -85,B 0,C 180,E1 14846.181,E2 14846.181} C_VEL
LIN {X 0,Y 455.569,Z 877.456,A -85,B 0,C 180,E1 14849.995,E2 14849.995} C_VEL
LIN {X 0,Y 455.662,Z 875.362,A -85,B 0,C 180,E1 14854.189,E2 14854.189} C_VEL
LIN {X 0,Y 456.493,Z 867.887,A -85,B 0,C 180,E1 14859.066,E2 14859.066} C_VEL
LIN {X 0,Y 458.317,Z 854.744,A -85,B 0,C 180,E1 14863.863,E2 14863.863} C_VEL
LIN {X 0,Y 461.296,Z 836.261,A -85,B 0,C 180,E1 14868.424,E2 14868.424} C_VEL
LIN {X 0,Y 465.68,Z 812.404,A -85,B 0,C 180,E1 14872.668,E2 14872.668} C_VEL
LIN {X 0,Y 470.705,Z 784.55,A -85,B 0,C 180,E1 14876.323,E2 14876.323} C_VEL
LIN {X 0,Y 476.18,Z 751.525,A -85,B 0,C 180,E1 14879.546,E2 14879.546} C_VEL
LIN {X 0,Y 481.261,Z 714.833,A -85,B 0,C 180,E1 14882.132,E2 14882.132} C_VEL
LIN {X 0,Y 484.371,Z 679.817,A -85,B 0,C 180,E1 14883.906,E2 14883.906} C_VEL
LIN {X 0,Y 476.723,Z 654.754,A -85,B 0,C 180,E1 14885.598,E2 14885.598} C_VEL
LIN {X 0,Y 459.425,Z 616.308,A -85,B 0,C 180,E1 14888.556,E2 14888.556} C_VEL
LIN {X 0,Y 452.405,Z 601.31,A -85,B 0,C 180,E1 14889.924,E2 14889.924} C_VEL
LIN {X 0,Y 452.247,Z 601.31,A -85,B 0,C 180,E1 14895.3,E2 14895.3} C_VEL
LIN {X 0,Y 452.263,Z 601.31,A -85,B 0,C 180,E1 14900.478,E2 14900.478} C_VEL
LIN {X 0,Y 452.341,Z 601.31,A -85,B 0,C 180,E1 14906.859,E2 14906.859} C_VEL
LIN {X 0,Y 452.701,Z 601.698,A -85,B 0,C 180,E1 14911.173,E2 14911.173} C_VEL
LIN {X 0,Y 473.02,Z 662.731,A -85,B 0,C 180,E1 14913.744,E2 14913.744} C_VEL
LIN {X 0,Y 470.902,Z 705.96,A -85,B 0,C 180,E1 14914.859,E2 14914.859} C_VEL
LIN {X 0,Y 467.997,Z 745.335,A -85,B 0,C 180,E1 14916.641,E2 14916.641} C_VEL
LIN {X 0,Y 464.624,Z 781.635,A -85,B 0,C 180,E1 14919.11,E2 14919.11} C_VEL
LIN {X 0,Y 461.577,Z 813.182,A -85,B 0,C 180,E1 14922.154,E2 14922.154} C_VEL
LIN {X 0,Y 458.946,Z 839.642,A -85,B 0,C 180,E1 14925.669,E2 14925.669} C_VEL
LIN {X 0,Y 457.275,Z 860.344,A -85,B 0,C 180,E1 14929.504,E2 14929.504} C_VEL
LIN {X 0,Y 456.426,Z 874.615,A -85,B 0,C 180,E1 14933.332,E2 14933.332} C_VEL
LIN {X 0,Y 456.217,Z 883.495,A -85,B 0,C 180,E1 14937.147,E2 14937.147} C_VEL
LIN {X 0,Y 456.254,Z 886.883,A -85,B 0,C 180,E1 14940.002,E2 14940.002} C_VEL
LIN {X 0,Y 456.849,Z 887.201,A -85,B 0,C 180,E1 14943.805,E2 14943.805} C_VEL
LIN {X 0,Y 458.208,Z 882.596,A -85,B 0,C 180,E1 14947.602,E2 14947.602} C_VEL
LIN {X 0,Y 460.374,Z 872.786,A -85,B 0,C 180,E1 14951.389,E2 14951.389} C_VEL
LIN {X 0,Y 463.336,Z 856.997,A -85,B 0,C 180,E1 14955.165,E2 14955.165} C_VEL
LIN {X 0,Y 467.348,Z 835.64,A -85,B 0,C 180,E1 14958.671,E2 14958.671} C_VEL
LIN {X 0,Y 472.363,Z 807.286,A -85,B 0,C 180,E1 14962.015,E2 14962.015} C_VEL
LIN {X 0,Y 478.158,Z 772.948,A -85,B 0,C 180,E1 14964.948,E2 14964.948} C_VEL
LIN {X 0,Y 484.643,Z 732.997,A -85,B 0,C 180,E1 14967.394,E2 14967.394} C_VEL
LIN {X 0,Y 491.398,Z 689.156,A -85,B 0,C 180,E1 14969.21,E2 14969.21} C_VEL
LIN {X 0,Y 492.997,Z 673.942,A -85,B 0,C 180,E1 14969.756,E2 14969.756} C_VEL
LIN {X 0,Y 487.903,Z 656.697,A -85,B 0,C 180,E1 14971.815,E2 14971.815} C_VEL
LIN {X 0,Y 483.601,Z 645.699,A -85,B 0,C 180,E1 14974.152,E2 14974.152} C_VEL
LIN {X 0,Y 481.852,Z 639.9,A -85,B 0,C 180,E1 14976.682,E2 14976.682} C_VEL
LIN {X 0,Y 482.329,Z 640.996,A -85,B 0,C 180,E1 14978.638,E2 14978.638} C_VEL
LIN {X 0,Y 485.423,Z 647.156,A -85,B 0,C 180,E1 14980.911,E2 14980.911} C_VEL
LIN {X 0,Y 490.824,Z 658.495,A -85,B 0,C 180,E1 14983.028,E2 14983.028} C_VEL
LIN {X 0,Y 496.619,Z 675.138,A -85,B 0,C 180,E1 14984.761,E2 14984.761} C_VEL
LIN {X 0,Y 500.921,Z 699.532,A -85,B 0,C 180,E1 14986.269,E2 14986.269} C_VEL
LIN {X 0,Y 495.318,Z 744.122,A -85,B 0,C 180,E1 14987.708,E2 14987.708} C_VEL
LIN {X 0,Y 488.535,Z 786.742,A -85,B 0,C 180,E1 14989.803,E2 14989.803} C_VEL
LIN {X 0,Y 481.132,Z 827.746,A -85,B 0,C 180,E1 14992.621,E2 14992.621} C_VEL
LIN {X 0,Y 473.975,Z 864.365,A -85,B 0,C 180,E1 14995.954,E2 14995.954} C_VEL
LIN {X 0,Y 467.04,Z 899.176,A -85,B 0,C 180,E1 15000.085,E2 15000.085} C_VEL
LIN {X 0,Y 461.474,Z 929.237,A -85,B 0,C 180,E1 15004.738,E2 15004.738} C_VEL
LIN {X 0,Y 457.621,Z 954.549,A -85,B 0,C 180,E1 15009.914,E2 15009.914} C_VEL
LIN {X 0,Y 455.533,Z 973.084,A -85,B 0,C 180,E1 15015.082,E2 15015.082} C_VEL
LIN {X 0,Y 454.824,Z 985.082,A -85,B 0,C 180,E1 15019.785,E2 15019.785} C_VEL
LIN {X 0,Y 454.714,Z 987.314,A -85,B 0,C 180,E1 15020.97,E2 15020.97} C_VEL
LIN {X 0,Y 452.178,Z 989.772,A -85,B 0,C 180,E1 15022.569,E2 15022.569} C_VEL
LIN {X 0,Y 446.874,Z 992.242,A -85,B 0,C 180,E1 15024.997,E2 15024.997} C_VEL
LIN {X 0,Y 446.781,Z 992.427,A -85,B 0,C 180,E1 15025.277,E2 15025.277} C_VEL
LIN {X 0,Y 447.007,Z 994.862,A -85,B 0,C 180,E1 15030.005,E2 15030.005} C_VEL
LIN {X 0,Y 446.852,Z 993.545,A -85,B 0,C 180,E1 15033.894,E2 15033.894} C_VEL
LIN {X 0,Y 446.746,Z 987.648,A -85,B 0,C 180,E1 15038.784,E2 15038.784} C_VEL
LIN {X 0,Y 447.367,Z 977.12,A -85,B 0,C 180,E1 15043.72,E2 15043.72} C_VEL
LIN {X 0,Y 449,Z 960.777,A -85,B 0,C 180,E1 15048.824,E2 15048.824} C_VEL
LIN {X 0,Y 452.219,Z 939.406,A -85,B 0,C 180,E1 15053.714,E2 15053.714} C_VEL
LIN {X 0,Y 457.379,Z 911.186,A -85,B 0,C 180,E1 15058.553,E2 15058.553} C_VEL
LIN {X 0,Y 463.607,Z 878.679,A -85,B 0,C 180,E1 15062.779,E2 15062.779} C_VEL
LIN {X 0,Y 470.78,Z 840.723,A -85,B 0,C 180,E1 15066.501,E2 15066.501} C_VEL
LIN {X 0,Y 477.823,Z 799.516,A -85,B 0,C 180,E1 15069.492,E2 15069.492} C_VEL
LIN {X 0,Y 484.054,Z 755.375,A -85,B 0,C 180,E1 15071.777,E2 15071.777} C_VEL
LIN {X 0,Y 488.686,Z 710.497,A -85,B 0,C 180,E1 15073.32,E2 15073.32} C_VEL
LIN {X 0,Y 488.908,Z 699.407,A -85,B 0,C 180,E1 15073.629,E2 15073.629} C_VEL
LIN {X 0,Y 454.156,Z 623.32,A -85,B 0,C 180,E1 15077.991,E2 15077.991} C_VEL
LIN {X 0,Y 444.403,Z 601.31,A -85,B 0,C 180,E1 15079.389,E2 15079.389} C_VEL
LIN {X 0,Y 444.469,Z 601.31,A -85,B 0,C 180,E1 15086.95,E2 15086.95} C_VEL
LIN {X 0,Y 444.677,Z 601.31,A -85,B 0,C 180,E1 15093.71,E2 15093.71} C_VEL
LIN {X 0,Y 444.997,Z 601.31,A -85,B 0,C 180,E1 15100.095,E2 15100.095} C_VEL
LIN {X 0,Y 445.236,Z 601.31,A -85,B 0,C 180,E1 15106.219,E2 15106.219} C_VEL
LIN {X 0,Y 445.597,Z 601.31,A -85,B 0,C 180,E1 15112.182,E2 15112.182} C_VEL
LIN {X 0,Y 445.967,Z 601.31,A -85,B 0,C 180,E1 15118.051,E2 15118.051} C_VEL
LIN {X 0,Y 445.879,Z 601.31,A -85,B 0,C 180,E1 15123.894,E2 15123.894} C_VEL
LIN {X 0,Y 445.494,Z 601.31,A -85,B 0,C 180,E1 15129.787,E2 15129.787} C_VEL
LIN {X 0,Y 445.186,Z 601.31,A -85,B 0,C 180,E1 15135.794,E2 15135.794} C_VEL
LIN {X 0,Y 444.914,Z 601.31,A -85,B 0,C 180,E1 15141.993,E2 15141.993} C_VEL
LIN {X 0,Y 444.617,Z 601.31,A -85,B 0,C 180,E1 15148.487,E2 15148.487} C_VEL
LIN {X 0,Y 444.441,Z 601.31,A -85,B 0,C 180,E1 15155.409,E2 15155.409} C_VEL
LIN {X 0,Y 444.316,Z 601.31,A -85,B 0,C 180,E1 15161.38,E2 15161.38} C_VEL
LIN {X 0,Y 444.372,Z 601.31,A -85,B 0,C 180,E1 15168.586,E2 15168.586} C_VEL
LIN {X 0,Y 444.443,Z 601.938,A -85,B 0,C 180,E1 15169.175,E2 15169.175} C_VEL
LIN {X 0,Y 466.365,Z 647.893,A -85,B 0,C 180,E1 15173.115,E2 15173.115} C_VEL
LIN {X 0,Y 477.47,Z 678.97,A -85,B 0,C 180,E1 15175.355,E2 15175.355} C_VEL
LIN {X 0,Y 477.674,Z 689.12,A -85,B 0,C 180,E1 15175.885,E2 15175.885} C_VEL
LIN {X 0,Y 473.235,Z 726.691,A -85,B 0,C 180,E1 15177.957,E2 15177.957} C_VEL
LIN {X 0,Y 467.703,Z 762.705,A -85,B 0,C 180,E1 15180.787,E2 15180.787} C_VEL
LIN {X 0,Y 462.149,Z 794.03,A -85,B 0,C 180,E1 15184.175,E2 15184.175} C_VEL
LIN {X 0,Y 456.897,Z 821.514,A -85,B 0,C 180,E1 15188.175,E2 15188.175} C_VEL
LIN {X 0,Y 452.544,Z 844.201,A -85,B 0,C 180,E1 15192.72,E2 15192.72} C_VEL
LIN {X 0,Y 449.918,Z 860.236,A -85,B 0,C 180,E1 15197.24,E2 15197.24} C_VEL
LIN {X 0,Y 448.317,Z 871.83,A -85,B 0,C 180,E1 15202.225,E2 15202.225} C_VEL
LIN {X 0,Y 447.784,Z 876.76,A -85,B 0,C 180,E1 15206.114,E2 15206.114} C_VEL
LIN {X 0,Y 447.742,Z 878.443,A -85,B 0,C 180,E1 15209.995,E2 15209.995} C_VEL
LIN {X 0,Y 447.89,Z 875.772,A -85,B 0,C 180,E1 15214.846,E2 15214.846} C_VEL
LIN {X 0,Y 448.809,Z 867.787,A -85,B 0,C 180,E1 15219.713,E2 15219.713} C_VEL
LIN {X 0,Y 450.94,Z 854.07,A -85,B 0,C 180,E1 15224.591,E2 15224.591} C_VEL
LIN {X 0,Y 454.283,Z 834.964,A -85,B 0,C 180,E1 15229.225,E2 15229.225} C_VEL
LIN {X 0,Y 459.107,Z 809.762,A -85,B 0,C 180,E1 15233.583,E2 15233.583} C_VEL
LIN {X 0,Y 464.738,Z 779.78,A -85,B 0,C 180,E1 15237.4,E2 15237.4} C_VEL
LIN {X 0,Y 470.293,Z 746.666,A -85,B 0,C 180,E1 15240.487,E2 15240.487} C_VEL
LIN {X 0,Y 475.299,Z 710.142,A -85,B 0,C 180,E1 15242.959,E2 15242.959} C_VEL
LIN {X 0,Y 477.764,Z 681.845,A -85,B 0,C 180,E1 15244.376,E2 15244.376} C_VEL
LIN {X 0,Y 468.648,Z 653.314,A -85,B 0,C 180,E1 15246.38,E2 15246.38} C_VEL
LIN {X 0,Y 451.203,Z 615.749,A -85,B 0,C 180,E1 15249.451,E2 15249.451} C_VEL
LIN {X 0,Y 444.474,Z 601.31,A -85,B 0,C 180,E1 15250.76,E2 15250.76} C_VEL
LIN {X 0,Y 444.289,Z 601.31,A -85,B 0,C 180,E1 15257.008,E2 15257.008} C_VEL
LIN {X 0,Y 444.307,Z 601.31,A -85,B 0,C 180,E1 15262.144,E2 15262.144} C_VEL
LIN {X 0,Y 444.482,Z 601.31,A -85,B 0,C 180,E1 15268.445,E2 15268.445} C_VEL
LIN {X 0,Y 444.747,Z 601.31,A -85,B 0,C 180,E1 15270.675,E2 15270.675} C_VEL
LIN {X 0,Y 465.559,Z 663.784,A -85,B 0,C 180,E1 15273.377,E2 15273.377} C_VEL
LIN {X 0,Y 463.469,Z 707.132,A -85,B 0,C 180,E1 15274.55,E2 15274.55} C_VEL
LIN {X 0,Y 460.478,Z 746.195,A -85,B 0,C 180,E1 15276.365,E2 15276.365} C_VEL
LIN {X 0,Y 457.009,Z 782.36,A -85,B 0,C 180,E1 15278.873,E2 15278.873} C_VEL
LIN {X 0,Y 453.96,Z 812.884,A -85,B 0,C 180,E1 15281.844,E2 15281.844} C_VEL
LIN {X 0,Y 451.249,Z 839.744,A -85,B 0,C 180,E1 15285.42,E2 15285.42} C_VEL
LIN {X 0,Y 449.496,Z 860.747,A -85,B 0,C 180,E1 15289.32,E2 15289.32} C_VEL
LIN {X 0,Y 448.587,Z 875.249,A -85,B 0,C 180,E1 15293.215,E2 15293.215} C_VEL
LIN {X 0,Y 448.381,Z 884.354,A -85,B 0,C 180,E1 15297.098,E2 15297.098} C_VEL
LIN {X 0,Y 448.422,Z 887.905,A -85,B 0,C 180,E1 15300.002,E2 15300.002} C_VEL
LIN {X 0,Y 449.094,Z 888.436,A -85,B 0,C 180,E1 15303.871,E2 15303.871} C_VEL
LIN {X 0,Y 450.52,Z 884.019,A -85,B 0,C 180,E1 15307.732,E2 15307.732} C_VEL
LIN {X 0,Y 452.81,Z 874.415,A -85,B 0,C 180,E1 15311.582,E2 15311.582} C_VEL
LIN {X 0,Y 456.19,Z 857.994,A -85,B 0,C 180,E1 15315.608,E2 15315.608} C_VEL
LIN {X 0,Y 460.549,Z 836.455,A -85,B 0,C 180,E1 15319.206,E2 15319.206} C_VEL
LIN {X 0,Y 465.92,Z 808.15,A -85,B 0,C 180,E1 15322.588,E2 15322.588} C_VEL
LIN {X 0,Y 472.262,Z 773.699,A -85,B 0,C 180,E1 15325.59,E2 15325.59} C_VEL
LIN {X 0,Y 479.371,Z 733.894,A -85,B 0,C 180,E1 15328.086,E2 15328.086} C_VEL
LIN {X 0,Y 486.44,Z 691.855,A -85,B 0,C 180,E1 15329.889,E2 15329.889} C_VEL
LIN {X 0,Y 488.212,Z 676.813,A -85,B 0,C 180,E1 15330.471,E2 15330.471} C_VEL
LIN {X 0,Y 484.062,Z 661.582,A -85,B 0,C 180,E1 15332.462,E2 15332.462} C_VEL
LIN {X 0,Y 480.831,Z 651.808,A -85,B 0,C 180,E1 15334.729,E2 15334.729} C_VEL
LIN {X 0,Y 479.904,Z 647.536,A -85,B 0,C 180,E1 15336.856,E2 15336.856} C_VEL
LIN {X 0,Y 480.385,Z 648.733,A -85,B 0,C 180,E1 15338.533,E2 15338.533} C_VEL
LIN {X 0,Y 483.289,Z 654.832,A -85,B 0,C 180,E1 15340.763,E2 15340.763} C_VEL
LIN {X 0,Y 488.044,Z 665.833,A -85,B 0,C 180,E1 15342.76,E2 15342.76} C_VEL
LIN {X 0,Y 493.034,Z 682.903,A -85,B 0,C 180,E1 15344.459,E2 15344.459} C_VEL
LIN {X 0,Y 495.494,Z 702.915,A -85,B 0,C 180,E1 15345.656,E2 15345.656} C_VEL
LIN {X 0,Y 488.855,Z 750.63,A -85,B 0,C 180,E1 15347.318,E2 15347.318} C_VEL
LIN {X 0,Y 481.167,Z 794.432,A -85,B 0,C 180,E1 15349.652,E2 15349.652} C_VEL
LIN {X 0,Y 472.655,Z 837.13,A -85,B 0,C 180,E1 15352.836,E2 15352.836} C_VEL
LIN {X 0,Y 464.684,Z 874.942,A -85,B 0,C 180,E1 15356.622,E2 15356.622} C_VEL
LIN {X 0,Y 457.631,Z 909.095,A -85,B 0,C 180,E1 15361.127,E2 15361.127} C_VEL
LIN {X 0,Y 452.424,Z 937.542,A -85,B 0,C 180,E1 15366.047,E2 15366.047} C_VEL
LIN {X 0,Y 448.849,Z 961.405,A -85,B 0,C 180,E1 15371.562,E2 15371.562} C_VEL
LIN {X 0,Y 447.234,Z 978.926,A -85,B 0,C 180,E1 15377.284,E2 15377.284} C_VEL
LIN {X 0,Y 446.845,Z 988.722,A -85,B 0,C 180,E1 15382.21,E2 15382.21} C_VEL
LIN {X 0,Y 446.781,Z 992.427,A -85,B 0,C 180,E1 15385.277,E2 15385.277} C_VEL
LIN {X 0,Y 445.538,Z 993.29,A -85,B 0,C 180,E1 15386.385,E2 15386.385} C_VEL
LIN {X 0,Y 439.185,Z 993.906,A -85,B 0,C 180,E1 15389.428,E2 15389.428} C_VEL
LIN {X 0,Y 439.134,Z 993.869,A -85,B 0,C 180,E1 15389.716,E2 15389.716} C_VEL
LIN {X 0,Y 438.997,Z 992.575,A -85,B 0,C 180,E1 15393.964,E2 15393.964} C_VEL
LIN {X 0,Y 438.894,Z 986.614,A -85,B 0,C 180,E1 15398.943,E2 15398.943} C_VEL
LIN {X 0,Y 439.526,Z 975.989,A -85,B 0,C 180,E1 15403.97,E2 15403.97} C_VEL
LIN {X 0,Y 441.351,Z 958.521,A -85,B 0,C 180,E1 15409.421,E2 15409.421} C_VEL
LIN {X 0,Y 444.905,Z 936.587,A -85,B 0,C 180,E1 15414.384,E2 15414.384} C_VEL
LIN {X 0,Y 449.782,Z 910.556,A -85,B 0,C 180,E1 15418.868,E2 15418.868} C_VEL
LIN {X 0,Y 456.293,Z 877.379,A -85,B 0,C 180,E1 15423.23,E2 15423.23} C_VEL
LIN {X 0,Y 463.53,Z 840.082,A -85,B 0,C 180,E1 15426.921,E2 15426.921} C_VEL
LIN {X 0,Y 470.712,Z 799.29,A -85,B 0,C 180,E1 15429.918,E2 15429.918} C_VEL
LIN {X 0,Y 477.175,Z 754.917,A -85,B 0,C 180,E1 15432.244,E2 15432.244} C_VEL
LIN {X 0,Y 482.01,Z 709.027,A -85,B 0,C 180,E1 15433.826,E2 15433.826} C_VEL
LIN {X 0,Y 481.837,Z 701.289,A -85,B 0,C 180,E1 15434.066,E2 15434.066} C_VEL
LIN {X 0,Y 448.392,Z 627.883,A -85,B 0,C 180,E1 15438.352,E2 15438.352} C_VEL
LIN {X 0,Y 436.449,Z 601.31,A -85,B 0,C 180,E1 15440.115,E2 15440.115} C_VEL
LIN {X 0,Y 436.505,Z 601.31,A -85,B 0,C 180,E1 15446.428,E2 15446.428} C_VEL
LIN {X 0,Y 436.731,Z 601.31,A -85,B 0,C 180,E1 15453.194,E2 15453.194} C_VEL
LIN {X 0,Y 437.039,Z 601.31,A -85,B 0,C 180,E1 15459.716,E2 15459.716} C_VEL
LIN {X 0,Y 437.314,Z 601.31,A -85,B 0,C 180,E1 15465.986,E2 15465.986} C_VEL
LIN {X 0,Y 437.675,Z 601.31,A -85,B 0,C 180,E1 15472.039,E2 15472.039} C_VEL
LIN {X 0,Y 438.071,Z 601.31,A -85,B 0,C 180,E1 15478.016,E2 15478.016} C_VEL
LIN {X 0,Y 437.982,Z 601.31,A -85,B 0,C 180,E1 15483.964,E2 15483.964} C_VEL
LIN {X 0,Y 437.562,Z 601.31,A -85,B 0,C 180,E1 15489.966,E2 15489.966} C_VEL
LIN {X 0,Y 437.247,Z 601.31,A -85,B 0,C 180,E1 15496.089,E2 15496.089} C_VEL
LIN {X 0,Y 437.005,Z 601.31,A -85,B 0,C 180,E1 15502.413,E2 15502.413} C_VEL
LIN {X 0,Y 436.632,Z 601.31,A -85,B 0,C 180,E1 15509.057,E2 15509.057} C_VEL
LIN {X 0,Y 436.532,Z 601.31,A -85,B 0,C 180,E1 15513.724,E2 15513.724} C_VEL
LIN {X 0,Y 436.409,Z 601.31,A -85,B 0,C 180,E1 15520.188,E2 15520.188} C_VEL
LIN {X 0,Y 436.398,Z 601.31,A -85,B 0,C 180,E1 15526.797,E2 15526.797} C_VEL
LIN {X 0,Y 436.424,Z 601.31,A -85,B 0,C 180,E1 15528.177,E2 15528.177} C_VEL
LIN {X 0,Y 441.381,Z 611.922,A -85,B 0,C 180,E1 15529.183,E2 15529.183} C_VEL
LIN {X 0,Y 460.388,Z 651.631,A -85,B 0,C 180,E1 15532.672,E2 15532.672} C_VEL
LIN {X 0,Y 471.061,Z 681.932,A -85,B 0,C 180,E1 15534.928,E2 15534.928} C_VEL
LIN {X 0,Y 470.205,Z 699.587,A -85,B 0,C 180,E1 15535.812,E2 15535.812} C_VEL
LIN {X 0,Y 465.317,Z 736.605,A -85,B 0,C 180,E1 15538.082,E2 15538.082} C_VEL
LIN {X 0,Y 459.872,Z 769.641,A -85,B 0,C 180,E1 15540.896,E2 15540.896} C_VEL
LIN {X 0,Y 454.091,Z 800.203,A -85,B 0,C 180,E1 15544.421,E2 15544.421} C_VEL
LIN {X 0,Y 448.838,Z 826.13,A -85,B 0,C 180,E1 15548.456,E2 15548.456} C_VEL
LIN {X 0,Y 444.604,Z 847.368,A -85,B 0,C 180,E1 15552.943,E2 15552.943} C_VEL
LIN {X 0,Y 442.054,Z 862.425,A -85,B 0,C 180,E1 15557.421,E2 15557.421} C_VEL
LIN {X 0,Y 440.552,Z 872.816,A -85,B 0,C 180,E1 15562.087,E2 15562.087} C_VEL
LIN {X 0,Y 439.847,Z 878.556,A -85,B 0,C 180,E1 15567.131,E2 15567.131} C_VEL
LIN {X 0,Y 439.917,Z 878.95,A -85,B 0,C 180,E1 15571.968,E2 15571.968} C_VEL
LIN {X 0,Y 440.388,Z 874.192,A -85,B 0,C 180,E1 15576.911,E2 15576.911} C_VEL
LIN {X 0,Y 441.739,Z 864.026,A -85,B 0,C 180,E1 15581.871,E2 15581.871} C_VEL
LIN {X 0,Y 444.493,Z 848.175,A -85,B 0,C 180,E1 15586.754,E2 15586.754} C_VEL
LIN {X 0,Y 448.66,Z 827.025,A -85,B 0,C 180,E1 15591.282,E2 15591.282} C_VEL
LIN {X 0,Y 453.991,Z 800.468,A -85,B 0,C 180,E1 15595.443,E2 15595.443} C_VEL
LIN {X 0,Y 459.781,Z 769.975,A -85,B 0,C 180,E1 15598.97,E2 15598.97} C_VEL
LIN {X 0,Y 465.365,Z 736.093,A -85,B 0,C 180,E1 15601.855,E2 15601.855} C_VEL
LIN {X 0,Y 470.26,Z 698.82,A -85,B 0,C 180,E1 15604.122,E2 15604.122} C_VEL
LIN {X 0,Y 470.944,Z 682.484,A -85,B 0,C 180,E1 15604.949,E2 15604.949} C_VEL
LIN {X 0,Y 460.256,Z 651.417,A -85,B 0,C 180,E1 15607.244,E2 15607.244} C_VEL
LIN {X 0,Y 443.371,Z 615.814,A -85,B 0,C 180,E1 15610.33,E2 15610.33} C_VEL
LIN {X 0,Y 436.467,Z 601.31,A -85,B 0,C 180,E1 15611.738,E2 15611.738} C_VEL
LIN {X 0,Y 436.369,Z 601.31,A -85,B 0,C 180,E1 15618.734,E2 15618.734} C_VEL
LIN {X 0,Y 436.384,Z 601.31,A -85,B 0,C 180,E1 15623.836,E2 15623.836} C_VEL
LIN {X 0,Y 436.777,Z 601.31,A -85,B 0,C 180,E1 15630.172,E2 15630.172} C_VEL
LIN {X 0,Y 458.109,Z 665.061,A -85,B 0,C 180,E1 15633.026,E2 15633.026} C_VEL
LIN {X 0,Y 456.071,Z 707.846,A -85,B 0,C 180,E1 15634.226,E2 15634.226} C_VEL
LIN {X 0,Y 452.95,Z 746.944,A -85,B 0,C 180,E1 15636.079,E2 15636.079} C_VEL
LIN {X 0,Y 449.389,Z 783.079,A -85,B 0,C 180,E1 15638.627,E2 15638.627} C_VEL
LIN {X 0,Y 446.127,Z 814.955,A -85,B 0,C 180,E1 15641.794,E2 15641.794} C_VEL
LIN {X 0,Y 443.392,Z 841.372,A -85,B 0,C 180,E1 15645.408,E2 15645.408} C_VEL
LIN {X 0,Y 441.624,Z 862.211,A -85,B 0,C 180,E1 15649.378,E2 15649.378} C_VEL
LIN {X 0,Y 440.704,Z 877.357,A -85,B 0,C 180,E1 15653.588,E2 15653.588} C_VEL
LIN {X 0,Y 440.535,Z 885.204,A -85,B 0,C 180,E1 15657.046,E2 15657.046} C_VEL
LIN {X 0,Y 440.602,Z 888.937,A -85,B 0,C 180,E1 15660.002,E2 15660.002} C_VEL
LIN {X 0,Y 441.324,Z 889.66,A -85,B 0,C 180,E1 15663.939,E2 15663.939} C_VEL
LIN {X 0,Y 442.835,Z 885.474,A -85,B 0,C 180,E1 15667.867,E2 15667.867} C_VEL
LIN {X 0,Y 445.265,Z 876.119,A -85,B 0,C 180,E1 15671.781,E2 15671.781} C_VEL
LIN {X 0,Y 448.86,Z 860.082,A -85,B 0,C 180,E1 15675.87,E2 15675.87} C_VEL
LIN {X 0,Y 453.44,Z 838.932,A -85,B 0,C 180,E1 15679.52,E2 15679.52} C_VEL
LIN {X 0,Y 459.333,Z 810.659,A -85,B 0,C 180,E1 15683.033,E2 15683.033} C_VEL
LIN {X 0,Y 466.454,Z 775.156,A -85,B 0,C 180,E1 15686.22,E2 15686.22} C_VEL
LIN {X 0,Y 474.39,Z 734.778,A -85,B 0,C 180,E1 15688.818,E2 15688.818} C_VEL
LIN {X 0,Y 482.221,Z 692.295,A -85,B 0,C 180,E1 15690.68,E2 15690.68} C_VEL
LIN {X 0,Y 483.821,Z 680.341,A -85,B 0,C 180,E1 15691.16,E2 15691.16} C_VEL
LIN {X 0,Y 480.476,Z 666.125,A -85,B 0,C 180,E1 15693.201,E2 15693.201} C_VEL
LIN {X 0,Y 478.17,Z 658.449,A -85,B 0,C 180,E1 15695.366,E2 15695.366} C_VEL
LIN {X 0,Y 478.003,Z 655.194,A -85,B 0,C 180,E1 15697.027,E2 15697.027} C_VEL
LIN {X 0,Y 478.474,Z 656.466,A -85,B 0,C 180,E1 15698.453,E2 15698.453} C_VEL
LIN {X 0,Y 481.1,Z 662.361,A -85,B 0,C 180,E1 15700.577,E2 15700.577} C_VEL
LIN {X 0,Y 485.219,Z 673.164,A -85,B 0,C 180,E1 15702.468,E2 15702.468} C_VEL
LIN {X 0,Y 489.136,Z 689.658,A -85,B 0,C 180,E1 15704.051,E2 15704.051} C_VEL
LIN {X 0,Y 490.509,Z 704.136,A -85,B 0,C 180,E1 15704.96,E2 15704.96} C_VEL
LIN {X 0,Y 483.397,Z 750.925,A -85,B 0,C 180,E1 15706.641,E2 15706.641} C_VEL
LIN {X 0,Y 475.034,Z 795.167,A -85,B 0,C 180,E1 15709.056,E2 15709.056} C_VEL
LIN {X 0,Y 466.334,Z 836.309,A -85,B 0,C 180,E1 15712.187,E2 15712.187} C_VEL
LIN {X 0,Y 457.837,Z 874.3,A -85,B 0,C 180,E1 15716.056,E2 15716.056} C_VEL
LIN {X 0,Y 450.515,Z 907.747,A -85,B 0,C 180,E1 15720.537,E2 15720.537} C_VEL
LIN {X 0,Y 444.862,Z 936.689,A -85,B 0,C 180,E1 15725.627,E2 15725.627} C_VEL
LIN {X 0,Y 441.197,Z 959.418,A -85,B 0,C 180,E1 15730.939,E2 15730.939} C_VEL
LIN {X 0,Y 439.51,Z 975.372,A -85,B 0,C 180,E1 15736.041,E2 15736.041} C_VEL
LIN {X 0,Y 438.97,Z 986.263,A -85,B 0,C 180,E1 15741.07,E2 15741.07} C_VEL
LIN {X 0,Y 438.976,Z 992.323,A -85,B 0,C 180,E1 15746.047,E2 15746.047} C_VEL
LIN {X 0,Y 439.134,Z 993.869,A -85,B 0,C 180,E1 15749.716,E2 15749.716} C_VEL
LIN {X 0,Y 436.746,Z 993.612,A -85,B 0,C 180,E1 15751.397,E2 15751.397} C_VEL
LIN {X 0,Y 431.141,Z 991.448,A -85,B 0,C 180,E1 15754.204,E2 15754.204} C_VEL
LIN {X 0,Y 431.042,Z 985.564,A -85,B 0,C 180,E1 15759.107,E2 15759.107} C_VEL
LIN {X 0,Y 431.724,Z 974.804,A -85,B 0,C 180,E1 15764.228,E2 15764.228} C_VEL
LIN {X 0,Y 433.643,Z 957.064,A -85,B 0,C 180,E1 15769.808,E2 15769.808} C_VEL
LIN {X 0,Y 437.449,Z 934.305,A -85,B 0,C 180,E1 15774.959,E2 15774.959} C_VEL
LIN {X 0,Y 442.847,Z 906.223,A -85,B 0,C 180,E1 15779.742,E2 15779.742} C_VEL
LIN {X 0,Y 449.384,Z 874.242,A -85,B 0,C 180,E1 15783.887,E2 15783.887} C_VEL
LIN {X 0,Y 456.513,Z 838.344,A -85,B 0,C 180,E1 15787.44,E2 15787.44} C_VEL
LIN {X 0,Y 463.645,Z 798.766,A -85,B 0,C 180,E1 15790.368,E2 15790.368} C_VEL
LIN {X 0,Y 470.265,Z 754.569,A -85,B 0,C 180,E1 15792.705,E2 15792.705} C_VEL
LIN {X 0,Y 475.208,Z 708.884,A -85,B 0,C 180,E1 15794.302,E2 15794.302} C_VEL
LIN {X 0,Y 474.462,Z 702.585,A -85,B 0,C 180,E1 15794.546,E2 15794.546} C_VEL
LIN {X 0,Y 442.548,Z 632.268,A -85,B 0,C 180,E1 15798.731,E2 15798.731} C_VEL
LIN {X 0,Y 428.497,Z 601.31,A -85,B 0,C 180,E1 15800.816,E2 15800.816} C_VEL
LIN {X 0,Y 428.642,Z 601.31,A -85,B 0,C 180,E1 15808.046,E2 15808.046} C_VEL
LIN {X 0,Y 428.897,Z 601.31,A -85,B 0,C 180,E1 15814.92,E2 15814.92} C_VEL
LIN {X 0,Y 429.17,Z 601.31,A -85,B 0,C 180,E1 15821.475,E2 15821.475} C_VEL
LIN {X 0,Y 429.463,Z 601.31,A -85,B 0,C 180,E1 15827.779,E2 15827.779} C_VEL
LIN {X 0,Y 429.918,Z 601.31,A -85,B 0,C 180,E1 15833.929,E2 15833.929} C_VEL
LIN {X 0,Y 430.325,Z 601.31,A -85,B 0,C 180,E1 15839.997,E2 15839.997} C_VEL
LIN {X 0,Y 429.925,Z 601.31,A -85,B 0,C 180,E1 15846.065,E2 15846.065} C_VEL
LIN {X 0,Y 429.523,Z 601.31,A -85,B 0,C 180,E1 15852.214,E2 15852.214} C_VEL
LIN {X 0,Y 429.186,Z 601.31,A -85,B 0,C 180,E1 15858.519,E2 15858.519} C_VEL
LIN {X 0,Y 428.885,Z 601.31,A -85,B 0,C 180,E1 15865.076,E2 15865.076} C_VEL
LIN {X 0,Y 428.627,Z 601.31,A -85,B 0,C 180,E1 15872.012,E2 15872.012} C_VEL
LIN {X 0,Y 428.51,Z 601.31,A -85,B 0,C 180,E1 15878.921,E2 15878.921} C_VEL
LIN {X 0,Y 428.486,Z 601.31,A -85,B 0,C 180,E1 15886.01,E2 15886.01} C_VEL
LIN {X 0,Y 428.509,Z 601.845,A -85,B 0,C 180,E1 15887.206,E2 15887.206} C_VEL
LIN {X 0,Y 450.754,Z 646.94,A -85,B 0,C 180,E1 15891.525,E2 15891.525} C_VEL
LIN {X 0,Y 463.107,Z 679.297,A -85,B 0,C 180,E1 15894.053,E2 15894.053} C_VEL
LIN {X 0,Y 464.866,Z 689.674,A -85,B 0,C 180,E1 15894.753,E2 15894.753} C_VEL
LIN {X 0,Y 460.111,Z 727.637,A -85,B 0,C 180,E1 15896.868,E2 15896.868} C_VEL
LIN {X 0,Y 454.323,Z 763.326,A -85,B 0,C 180,E1 15899.7,E2 15899.7} C_VEL
LIN {X 0,Y 448.295,Z 794.569,A -85,B 0,C 180,E1 15903.118,E2 15903.118} C_VEL
LIN {X 0,Y 442.682,Z 821.509,A -85,B 0,C 180,E1 15907.082,E2 15907.082} C_VEL
LIN {X 0,Y 437.993,Z 844.076,A -85,B 0,C 180,E1 15911.593,E2 15911.593} C_VEL
LIN {X 0,Y 434.767,Z 861.217,A -85,B 0,C 180,E1 15916.44,E2 15916.44} C_VEL
LIN {X 0,Y 433.051,Z 871.958,A -85,B 0,C 180,E1 15920.935,E2 15920.935} C_VEL
LIN {X 0,Y 432.152,Z 878.733,A -85,B 0,C 180,E1 15925.973,E2 15925.973} C_VEL
LIN {X 0,Y 432.081,Z 880.417,A -85,B 0,C 180,E1 15929.994,E2 15929.994} C_VEL
LIN {X 0,Y 432.267,Z 877.747,A -85,B 0,C 180,E1 15935.022,E2 15935.022} C_VEL
LIN {X 0,Y 433.313,Z 869.766,A -85,B 0,C 180,E1 15940.064,E2 15940.064} C_VEL
LIN {X 0,Y 435.713,Z 856.059,A -85,B 0,C 180,E1 15945.113,E2 15945.113} C_VEL
LIN {X 0,Y 439.444,Z 836.934,A -85,B 0,C 180,E1 15949.901,E2 15949.901} C_VEL
LIN {X 0,Y 444.729,Z 811.766,A -85,B 0,C 180,E1 15954.387,E2 15954.387} C_VEL
LIN {X 0,Y 450.793,Z 781.962,A -85,B 0,C 180,E1 15958.288,E2 15958.288} C_VEL
LIN {X 0,Y 456.851,Z 748.495,A -85,B 0,C 180,E1 15961.485,E2 15961.485} C_VEL
LIN {X 0,Y 462.174,Z 712.174,A -85,B 0,C 180,E1 15964,E2 15964} C_VEL
LIN {X 0,Y 464.551,Z 685.323,A -85,B 0,C 180,E1 15965.393,E2 15965.393} C_VEL
LIN {X 0,Y 453.743,Z 653.746,A -85,B 0,C 180,E1 15967.808,E2 15967.808} C_VEL
LIN {X 0,Y 435.98,Z 616.542,A -85,B 0,C 180,E1 15971.177,E2 15971.177} C_VEL
LIN {X 0,Y 428.546,Z 601.995,A -85,B 0,C 180,E1 15972.673,E2 15972.673} C_VEL
LIN {X 0,Y 428.442,Z 601.31,A -85,B 0,C 180,E1 15977.951,E2 15977.951} C_VEL
LIN {X 0,Y 428.475,Z 601.31,A -85,B 0,C 180,E1 15984.414,E2 15984.414} C_VEL
LIN {X 0,Y 428.836,Z 601.979,A -85,B 0,C 180,E1 15989.7,E2 15989.7} C_VEL
LIN {X 0,Y 450.85,Z 667.047,A -85,B 0,C 180,E1 15992.693,E2 15992.693} C_VEL
LIN {X 0,Y 448.542,Z 710.304,A -85,B 0,C 180,E1 15993.959,E2 15993.959} C_VEL
LIN {X 0,Y 445.273,Z 749.701,A -85,B 0,C 180,E1 15995.907,E2 15995.907} C_VEL
LIN {X 0,Y 441.675,Z 785.211,A -85,B 0,C 180,E1 15998.499,E2 15998.499} C_VEL
LIN {X 0,Y 438.301,Z 816.964,A -85,B 0,C 180,E1 16001.742,E2 16001.742} C_VEL
LIN {X 0,Y 435.561,Z 842.96,A -85,B 0,C 180,E1 16005.398,E2 16005.398} C_VEL
LIN {X 0,Y 433.782,Z 863.651,A -85,B 0,C 180,E1 16009.438,E2 16009.438} C_VEL
LIN {X 0,Y 432.865,Z 877.988,A -85,B 0,C 180,E1 16013.472,E2 16013.472} C_VEL
LIN {X 0,Y 432.689,Z 886.372,A -85,B 0,C 180,E1 16017.179,E2 16017.179} C_VEL
LIN {X 0,Y 432.795,Z 889.952,A -85,B 0,C 180,E1 16020.003,E2 16020.003} C_VEL
LIN {X 0,Y 433.547,Z 890.904,A -85,B 0,C 180,E1 16024.01,E2 16024.01} C_VEL
LIN {X 0,Y 435.154,Z 886.925,A -85,B 0,C 180,E1 16028.007,E2 16028.007} C_VEL
LIN {X 0,Y 437.745,Z 877.823,A -85,B 0,C 180,E1 16031.987,E2 16031.987} C_VEL
LIN {X 0,Y 441.499,Z 862.462,A -85,B 0,C 180,E1 16036.085,E2 16036.085} C_VEL
LIN {X 0,Y 446.413,Z 841.602,A -85,B 0,C 180,E1 16039.84,E2 16039.84} C_VEL
LIN {X 0,Y 452.786,Z 813.322,A -85,B 0,C 180,E1 16043.484,E2 16043.484} C_VEL
LIN {X 0,Y 460.512,Z 778.266,A -85,B 0,C 180,E1 16046.763,E2 16046.763} C_VEL
LIN {X 0,Y 469.332,Z 737.544,A -85,B 0,C 180,E1 16049.49,E2 16049.49} C_VEL
LIN {X 0,Y 477.871,Z 695.595,A -85,B 0,C 180,E1 16051.408,E2 16051.408} C_VEL
LIN {X 0,Y 479.732,Z 683.878,A -85,B 0,C 180,E1 16051.891,E2 16051.891} C_VEL
LIN {X 0,Y 477.333,Z 671.512,A -85,B 0,C 180,E1 16053.865,E2 16053.865} C_VEL
LIN {X 0,Y 475.97,Z 665.434,A -85,B 0,C 180,E1 16055.771,E2 16055.771} C_VEL
LIN {X 0,Y 476.159,Z 662.882,A -85,B 0,C 180,E1 16057.303,E2 16057.303} C_VEL
LIN {X 0,Y 476.84,Z 665.185,A -85,B 0,C 180,E1 16058.79,E2 16058.79} C_VEL
LIN {X 0,Y 479.232,Z 670.735,A -85,B 0,C 180,E1 16060.579,E2 16060.579} C_VEL
LIN {X 0,Y 482.8,Z 682.494,A -85,B 0,C 180,E1 16062.396,E2 16062.396} C_VEL
LIN {X 0,Y 485.261,Z 698.744,A -85,B 0,C 180,E1 16063.792,E2 16063.792} C_VEL
LIN {X 0,Y 485.358,Z 708.401,A -85,B 0,C 180,E1 16064.326,E2 16064.326} C_VEL
LIN {X 0,Y 477.594,Z 753.953,A -85,B 0,C 180,E1 16066.059,E2 16066.059} C_VEL
LIN {X 0,Y 469.072,Z 795.919,A -85,B 0,C 180,E1 16068.432,E2 16068.432} C_VEL
LIN {X 0,Y 459.594,Z 837.755,A -85,B 0,C 180,E1 16071.71,E2 16071.71} C_VEL
LIN {X 0,Y 450.788,Z 874.907,A -85,B 0,C 180,E1 16075.611,E2 16075.611} C_VEL
LIN {X 0,Y 443.173,Z 907.65,A -85,B 0,C 180,E1 16080.114,E2 16080.114} C_VEL
LIN {X 0,Y 437.443,Z 935.193,A -85,B 0,C 180,E1 16085.044,E2 16085.044} C_VEL
LIN {X 0,Y 433.384,Z 958.964,A -85,B 0,C 180,E1 16090.703,E2 16090.703} C_VEL
LIN {X 0,Y 431.589,Z 975.783,A -85,B 0,C 180,E1 16096.298,E2 16096.298} C_VEL
LIN {X 0,Y 431.102,Z 985.361,A -85,B 0,C 180,E1 16100.905,E2 16100.905} C_VEL
LIN {X 0,Y 431.122,Z 991.407,A -85,B 0,C 180,E1 16105.975,E2 16105.975} C_VEL
LIN {X 0,Y 431.358,Z 993,A -85,B 0,C 180,E1 16110.006,E2 16110.006} C_VEL
LIN {X 0,Y 431.141,Z 991.448,A -85,B 0,C 180,E1 16114.204,E2 16114.204} C_VEL
LIN {X 0,Y 428.515,Z 989.675,A -85,B 0,C 180,E1 16115.903,E2 16115.903} C_VEL
LIN {X 0,Y 423.264,Z 985.843,A -85,B 0,C 180,E1 16118.437,E2 16118.437} C_VEL
LIN {X 0,Y 423.179,Z 985.361,A -85,B 0,C 180,E1 16118.729,E2 16118.729} C_VEL
LIN {X 0,Y 423.786,Z 974.893,A -85,B 0,C 180,E1 16123.971,E2 16123.971} C_VEL
LIN {X 0,Y 425.459,Z 959.189,A -85,B 0,C 180,E1 16129.187,E2 16129.187} C_VEL
LIN {X 0,Y 429.137,Z 937.094,A -85,B 0,C 180,E1 16134.517,E2 16134.517} C_VEL
LIN {X 0,Y 434.524,Z 909.591,A -85,B 0,C 180,E1 16139.46,E2 16139.46} C_VEL
LIN {X 0,Y 441.392,Z 876.51,A -85,B 0,C 180,E1 16143.947,E2 16143.947} C_VEL
LIN {X 0,Y 449.021,Z 839.174,A -85,B 0,C 180,E1 16147.744,E2 16147.744} C_VEL
LIN {X 0,Y 456.549,Z 798.563,A -85,B 0,C 180,E1 16150.804,E2 16150.804} C_VEL
LIN {X 0,Y 463.266,Z 754.946,A -85,B 0,C 180,E1 16153.151,E2 16153.151} C_VEL
LIN {X 0,Y 468.461,Z 708.273,A -85,B 0,C 180,E1 16154.8,E2 16154.8} C_VEL
LIN {X 0,Y 447.256,Z 659.431,A -85,B 0,C 180,E1 16157.684,E2 16157.684} C_VEL
LIN {X 0,Y 420.578,Z 601.31,A -85,B 0,C 180,E1 16161.511,E2 16161.511} C_VEL
LIN {X 0,Y 420.613,Z 601.31,A -85,B 0,C 180,E1 16167.297,E2 16167.297} C_VEL
LIN {X 0,Y 420.904,Z 601.31,A -85,B 0,C 180,E1 16174.409,E2 16174.409} C_VEL
LIN {X 0,Y 421.22,Z 601.31,A -85,B 0,C 180,E1 16181.112,E2 16181.112} C_VEL
LIN {X 0,Y 421.523,Z 601.31,A -85,B 0,C 180,E1 16187.545,E2 16187.545} C_VEL
LIN {X 0,Y 422.02,Z 601.31,A -85,B 0,C 180,E1 16193.815,E2 16193.815} C_VEL
LIN {X 0,Y 422.437,Z 601.31,A -85,B 0,C 180,E1 16199.997,E2 16199.997} C_VEL
LIN {X 0,Y 422.026,Z 601.31,A -85,B 0,C 180,E1 16206.179,E2 16206.179} C_VEL
LIN {X 0,Y 421.586,Z 601.31,A -85,B 0,C 180,E1 16212.448,E2 16212.448} C_VEL
LIN {X 0,Y 421.237,Z 601.31,A -85,B 0,C 180,E1 16218.882,E2 16218.882} C_VEL
LIN {X 0,Y 420.892,Z 601.31,A -85,B 0,C 180,E1 16225.586,E2 16225.586} C_VEL
LIN {X 0,Y 420.619,Z 601.31,A -85,B 0,C 180,E1 16232.696,E2 16232.696} C_VEL
LIN {X 0,Y 420.56,Z 601.31,A -85,B 0,C 180,E1 16237.756,E2 16237.756} C_VEL
LIN {X 0,Y 420.429,Z 601.31,A -85,B 0,C 180,E1 16243.872,E2 16243.872} C_VEL
LIN {X 0,Y 420.631,Z 602.085,A -85,B 0,C 180,E1 16246.155,E2 16246.155} C_VEL
LIN {X 0,Y 443.032,Z 646.494,A -85,B 0,C 180,E1 16250.677,E2 16250.677} C_VEL
LIN {X 0,Y 456.249,Z 680.553,A -85,B 0,C 180,E1 16253.454,E2 16253.454} C_VEL
LIN {X 0,Y 458.473,Z 690.344,A -85,B 0,C 180,E1 16254.187,E2 16254.187} C_VEL
LIN {X 0,Y 453.645,Z 727.96,A -85,B 0,C 180,E1 16256.286,E2 16256.286} C_VEL
LIN {X 0,Y 447.786,Z 762.906,A -85,B 0,C 180,E1 16259.069,E2 16259.069} C_VEL
LIN {X 0,Y 441.287,Z 795.549,A -85,B 0,C 180,E1 16262.656,E2 16262.656} C_VEL
LIN {X 0,Y 435.441,Z 822.486,A -85,B 0,C 180,E1 16266.677,E2 16266.677} C_VEL
LIN {X 0,Y 430.52,Z 845.075,A -85,B 0,C 180,E1 16271.262,E2 16271.262} C_VEL
LIN {X 0,Y 427.142,Z 862.066,A -85,B 0,C 180,E1 16276.141,E2 16276.141} C_VEL
LIN {X 0,Y 425.293,Z 872.949,A -85,B 0,C 180,E1 16280.769,E2 16280.769} C_VEL
LIN {X 0,Y 424.347,Z 879.72,A -85,B 0,C 180,E1 16285.899,E2 16285.899} C_VEL
LIN {X 0,Y 424.214,Z 881.242,A -85,B 0,C 180,E1 16291.017,E2 16291.017} C_VEL
LIN {X 0,Y 424.62,Z 877.569,A -85,B 0,C 180,E1 16296.14,E2 16296.14} C_VEL
LIN {X 0,Y 425.932,Z 868.655,A -85,B 0,C 180,E1 16301.234,E2 16301.234} C_VEL
LIN {X 0,Y 428.756,Z 853.555,A -85,B 0,C 180,E1 16306.417,E2 16306.417} C_VEL
LIN {X 0,Y 433.089,Z 833.221,A -85,B 0,C 180,E1 16311.222,E2 16311.222} C_VEL
LIN {X 0,Y 438.622,Z 807.92,A -85,B 0,C 180,E1 16315.545,E2 16315.545} C_VEL
LIN {X 0,Y 444.711,Z 778.7,A -85,B 0,C 180,E1 16319.232,E2 16319.232} C_VEL
LIN {X 0,Y 450.978,Z 744.984,A -85,B 0,C 180,E1 16322.37,E2 16322.37} C_VEL
LIN {X 0,Y 456.257,Z 708.832,A -85,B 0,C 180,E1 16324.777,E2 16324.777} C_VEL
LIN {X 0,Y 458.054,Z 687.429,A -85,B 0,C 180,E1 16325.901,E2 16325.901} C_VEL
LIN {X 0,Y 446.848,Z 655.137,A -85,B 0,C 180,E1 16328.466,E2 16328.466} C_VEL
LIN {X 0,Y 428.853,Z 617.693,A -85,B 0,C 180,E1 16332.015,E2 16332.015} C_VEL
LIN {X 0,Y 420.736,Z 602.704,A -85,B 0,C 180,E1 16333.693,E2 16333.693} C_VEL
LIN {X 0,Y 420.595,Z 601.31,A -85,B 0,C 180,E1 16333.92,E2 16333.92} C_VEL
LIN {X 0,Y 420.449,Z 601.31,A -85,B 0,C 180,E1 16339.572,E2 16339.572} C_VEL
LIN {X 0,Y 420.562,Z 601.31,A -85,B 0,C 180,E1 16345.95,E2 16345.95} C_VEL
LIN {X 0,Y 420.83,Z 601.31,A -85,B 0,C 180,E1 16349.158,E2 16349.158} C_VEL
LIN {X 0,Y 443.703,Z 669.422,A -85,B 0,C 180,E1 16352.364,E2 16352.364} C_VEL
LIN {X 0,Y 441.14,Z 711.318,A -85,B 0,C 180,E1 16353.626,E2 16353.626} C_VEL
LIN {X 0,Y 437.751,Z 750.449,A -85,B 0,C 180,E1 16355.602,E2 16355.602} C_VEL
LIN {X 0,Y 434.074,Z 785.866,A -85,B 0,C 180,E1 16358.238,E2 16358.238} C_VEL
LIN {X 0,Y 430.597,Z 817.679,A -85,B 0,C 180,E1 16361.544,E2 16361.544} C_VEL
LIN {X 0,Y 427.699,Z 844.516,A -85,B 0,C 180,E1 16365.385,E2 16365.385} C_VEL
LIN {X 0,Y 425.917,Z 865.079,A -85,B 0,C 180,E1 16369.5,E2 16369.5} C_VEL
LIN {X 0,Y 425.024,Z 880.005,A -85,B 0,C 180,E1 16373.864,E2 16373.864} C_VEL
LIN {X 0,Y 424.9,Z 888.5,A -85,B 0,C 180,E1 16377.959,E2 16377.959} C_VEL
LIN {X 0,Y 425.158,Z 892.146,A -85,B 0,C 180,E1 16382.045,E2 16382.045} C_VEL
LIN {X 0,Y 426.587,Z 890.87,A -85,B 0,C 180,E1 16386.118,E2 16386.118} C_VEL
LIN {X 0,Y 428.698,Z 884.691,A -85,B 0,C 180,E1 16390.179,E2 16390.179} C_VEL
LIN {X 0,Y 431.999,Z 873.193,A -85,B 0,C 180,E1 16394.212,E2 16394.212} C_VEL
LIN {X 0,Y 436.463,Z 855.665,A -85,B 0,C 180,E1 16398.205,E2 16398.205} C_VEL
LIN {X 0,Y 442.797,Z 830.97,A -85,B 0,C 180,E1 16402.109,E2 16402.109} C_VEL
LIN {X 0,Y 450.271,Z 799.846,A -85,B 0,C 180,E1 16405.671,E2 16405.671} C_VEL
LIN {X 0,Y 459.537,Z 761.386,A -85,B 0,C 180,E1 16408.853,E2 16408.853} C_VEL
LIN {X 0,Y 469.401,Z 719.414,A -85,B 0,C 180,E1 16411.294,E2 16411.294} C_VEL
LIN {X 0,Y 475.984,Z 687.421,A -85,B 0,C 180,E1 16412.677,E2 16412.677} C_VEL
LIN {X 0,Y 474.463,Z 676.357,A -85,B 0,C 180,E1 16414.695,E2 16414.695} C_VEL
LIN {X 0,Y 474.227,Z 670.635,A -85,B 0,C 180,E1 16417.099,E2 16417.099} C_VEL
LIN {X 0,Y 474.779,Z 672.482,A -85,B 0,C 180,E1 16418.523,E2 16418.523} C_VEL
LIN {X 0,Y 476.879,Z 678.113,A -85,B 0,C 180,E1 16420.317,E2 16420.317} C_VEL
LIN {X 0,Y 479.644,Z 689.419,A -85,B 0,C 180,E1 16422.02,E2 16422.02} C_VEL
LIN {X 0,Y 481.176,Z 707.171,A -85,B 0,C 180,E1 16423.477,E2 16423.477} C_VEL
LIN {X 0,Y 472.593,Z 754.134,A -85,B 0,C 180,E1 16425.311,E2 16425.311} C_VEL
LIN {X 0,Y 463.147,Z 797.215,A -85,B 0,C 180,E1 16427.812,E2 16427.812} C_VEL
LIN {X 0,Y 453.435,Z 837.314,A -85,B 0,C 180,E1 16431.031,E2 16431.031} C_VEL
LIN {X 0,Y 444.237,Z 873.847,A -85,B 0,C 180,E1 16434.931,E2 16434.931} C_VEL
LIN {X 0,Y 436.182,Z 906.378,A -85,B 0,C 180,E1 16439.474,E2 16439.474} C_VEL
LIN {X 0,Y 429.881,Z 934.532,A -85,B 0,C 180,E1 16444.61,E2 16444.61} C_VEL
LIN {X 0,Y 425.662,Z 958.09,A -85,B 0,C 180,E1 16450.339,E2 16450.339} C_VEL
LIN {X 0,Y 423.744,Z 974.889,A -85,B 0,C 180,E1 16456.039,E2 16456.039} C_VEL
LIN {X 0,Y 423.226,Z 984.466,A -85,B 0,C 180,E1 16460.735,E2 16460.735} C_VEL
LIN {X 0,Y 423.279,Z 990.49,A -85,B 0,C 180,E1 16465.9,E2 16465.9} C_VEL
LIN {X 0,Y 423.512,Z 992.051,A -85,B 0,C 180,E1 16470.006,E2 16470.006} C_VEL
LIN {X 0,Y 423.305,Z 990.547,A -85,B 0,C 180,E1 16474.167,E2 16474.167} C_VEL
LIN {X 0,Y 423.179,Z 985.361,A -85,B 0,C 180,E1 16478.729,E2 16478.729} C_VEL
LIN {X 0,Y 420.829,Z 982.297,A -85,B 0,C 180,E1 16480.432,E2 16480.432} C_VEL
LIN {X 0,Y 415.835,Z 975.965,A -85,B 0,C 180,E1 16483.25,E2 16483.25} C_VEL
LIN {X 0,Y 417.265,Z 961.328,A -85,B 0,C 180,E1 16488.532,E2 16488.532} C_VEL
LIN {X 0,Y 420.904,Z 939.198,A -85,B 0,C 180,E1 16494.179,E2 16494.179} C_VEL
LIN {X 0,Y 426.623,Z 910.667,A -85,B 0,C 180,E1 16499.517,E2 16499.517} C_VEL
LIN {X 0,Y 433.753,Z 877.104,A -85,B 0,C 180,E1 16504.185,E2 16504.185} C_VEL
LIN {X 0,Y 441.74,Z 839.062,A -85,B 0,C 180,E1 16508.134,E2 16508.134} C_VEL
LIN {X 0,Y 449.489,Z 798.032,A -85,B 0,C 180,E1 16511.264,E2 16511.264} C_VEL
LIN {X 0,Y 456.354,Z 754.419,A -85,B 0,C 180,E1 16513.634,E2 16513.634} C_VEL
LIN {X 0,Y 461.037,Z 708.418,A -85,B 0,C 180,E1 16515.326,E2 16515.326} C_VEL
LIN {X 0,Y 434.051,Z 648.065,A -85,B 0,C 180,E1 16519.04,E2 16519.04} C_VEL
LIN {X 0,Y 412.653,Z 601.31,A -85,B 0,C 180,E1 16522.277,E2 16522.277} C_VEL
LIN {X 0,Y 412.738,Z 601.31,A -85,B 0,C 180,E1 16529.077,E2 16529.077} C_VEL
LIN {X 0,Y 413.095,Z 601.31,A -85,B 0,C 180,E1 16536.207,E2 16536.207} C_VEL
LIN {X 0,Y 413.385,Z 601.31,A -85,B 0,C 180,E1 16542.95,E2 16542.95} C_VEL
LIN {X 0,Y 413.736,Z 601.31,A -85,B 0,C 180,E1 16549.448,E2 16549.448} C_VEL
LIN {X 0,Y 414.259,Z 601.31,A -85,B 0,C 180,E1 16555.803,E2 16555.803} C_VEL
LIN {X 0,Y 414.441,Z 601.31,A -85,B 0,C 180,E1 16562.092,E2 16562.092} C_VEL
LIN {X 0,Y 413.869,Z 601.31,A -85,B 0,C 180,E1 16568.664,E2 16568.664} C_VEL
LIN {X 0,Y 413.546,Z 601.31,A -85,B 0,C 180,E1 16574.855,E2 16574.855} C_VEL
LIN {X 0,Y 413.217,Z 601.31,A -85,B 0,C 180,E1 16581.504,E2 16581.504} C_VEL
LIN {X 0,Y 412.866,Z 601.31,A -85,B 0,C 180,E1 16588.486,E2 16588.486} C_VEL
LIN {X 0,Y 412.694,Z 601.31,A -85,B 0,C 180,E1 16593.406,E2 16593.406} C_VEL
LIN {X 0,Y 412.533,Z 601.31,A -85,B 0,C 180,E1 16599.519,E2 16599.519} C_VEL
LIN {X 0,Y 412.543,Z 601.647,A -85,B 0,C 180,E1 16604.981,E2 16604.981} C_VEL
LIN {X 0,Y 415.206,Z 607.17,A -85,B 0,C 180,E1 16605.601,E2 16605.601} C_VEL
LIN {X 0,Y 434.137,Z 643.695,A -85,B 0,C 180,E1 16609.56,E2 16609.56} C_VEL
LIN {X 0,Y 448.91,Z 680.121,A -85,B 0,C 180,E1 16612.702,E2 16612.702} C_VEL
LIN {X 0,Y 451.955,Z 692.517,A -85,B 0,C 180,E1 16613.668,E2 16613.668} C_VEL
LIN {X 0,Y 446.884,Z 730.63,A -85,B 0,C 180,E1 16615.854,E2 16615.854} C_VEL
LIN {X 0,Y 440.585,Z 766.515,A -85,B 0,C 180,E1 16618.795,E2 16618.795} C_VEL
LIN {X 0,Y 433.92,Z 798.429,A -85,B 0,C 180,E1 16622.434,E2 16622.434} C_VEL
LIN {X 0,Y 427.878,Z 824.95,A -85,B 0,C 180,E1 16626.517,E2 16626.517} C_VEL
LIN {X 0,Y 422.801,Z 847.095,A -85,B 0,C 180,E1 16631.178,E2 16631.178} C_VEL
LIN {X 0,Y 419.493,Z 863.061,A -85,B 0,C 180,E1 16635.883,E2 16635.883} C_VEL
LIN {X 0,Y 417.528,Z 873.943,A -85,B 0,C 180,E1 16640.595,E2 16640.595} C_VEL
LIN {X 0,Y 416.529,Z 880.709,A -85,B 0,C 180,E1 16645.822,E2 16645.822} C_VEL
LIN {X 0,Y 416.423,Z 882.391,A -85,B 0,C 180,E1 16649.994,E2 16649.994} C_VEL
LIN {X 0,Y 416.649,Z 879.723,A -85,B 0,C 180,E1 16655.211,E2 16655.211} C_VEL
LIN {X 0,Y 417.831,Z 871.753,A -85,B 0,C 180,E1 16660.441,E2 16660.441} C_VEL
LIN {X 0,Y 420.498,Z 858.062,A -85,B 0,C 180,E1 16665.673,E2 16665.673} C_VEL
LIN {X 0,Y 424.674,Z 838.91,A -85,B 0,C 180,E1 16670.624,E2 16670.624} C_VEL
LIN {X 0,Y 430.058,Z 815.315,A -85,B 0,C 180,E1 16675.005,E2 16675.005} C_VEL
LIN {X 0,Y 436.626,Z 785.702,A -85,B 0,C 180,E1 16679.061,E2 16679.061} C_VEL
LIN {X 0,Y 443.011,Z 753.303,A -85,B 0,C 180,E1 16682.298,E2 16682.298} C_VEL
LIN {X 0,Y 448.808,Z 717.066,A -85,B 0,C 180,E1 16684.927,E2 16684.927} C_VEL
LIN {X 0,Y 451.619,Z 690.063,A -85,B 0,C 180,E1 16686.39,E2 16686.39} C_VEL
LIN {X 0,Y 440.321,Z 657.397,A -85,B 0,C 180,E1 16689.082,E2 16689.082} C_VEL
LIN {X 0,Y 423.3,Z 622.132,A -85,B 0,C 180,E1 16692.551,E2 16692.551} C_VEL
LIN {X 0,Y 412.605,Z 602.144,A -85,B 0,C 180,E1 16694.872,E2 16694.872} C_VEL
LIN {X 0,Y 412.531,Z 601.31,A -85,B 0,C 180,E1 16695.76,E2 16695.76} C_VEL
LIN {X 0,Y 412.489,Z 601.31,A -85,B 0,C 180,E1 16701.37,E2 16701.37} C_VEL
LIN {X 0,Y 412.896,Z 601.31,A -85,B 0,C 180,E1 16708.614,E2 16708.614} C_VEL
LIN {X 0,Y 436.208,Z 670.296,A -85,B 0,C 180,E1 16711.963,E2 16711.963} C_VEL
LIN {X 0,Y 433.731,Z 712.118,A -85,B 0,C 180,E1 16713.28,E2 16713.28} C_VEL
LIN {X 0,Y 430.236,Z 750.953,A -85,B 0,C 180,E1 16715.287,E2 16715.287} C_VEL
LIN {X 0,Y 426.409,Z 786.858,A -85,B 0,C 180,E1 16718.007,E2 16718.007} C_VEL
LIN {X 0,Y 422.854,Z 818.919,A -85,B 0,C 180,E1 16721.408,E2 16721.408} C_VEL
LIN {X 0,Y 419.851,Z 846.031,A -85,B 0,C 180,E1 16725.373,E2 16725.373} C_VEL
LIN {X 0,Y 418.043,Z 866.489,A -85,B 0,C 180,E1 16729.564,E2 16729.564} C_VEL
LIN {X 0,Y 417.182,Z 880.625,A -85,B 0,C 180,E1 16733.749,E2 16733.749} C_VEL
LIN {X 0,Y 417.059,Z 889.365,A -85,B 0,C 180,E1 16737.921,E2 16737.921} C_VEL
LIN {X 0,Y 417.359,Z 893.256,A -85,B 0,C 180,E1 16742.083,E2 16742.083} C_VEL
LIN {X 0,Y 418.86,Z 892.229,A -85,B 0,C 180,E1 16746.232,E2 16746.232} C_VEL
LIN {X 0,Y 421.09,Z 886.314,A -85,B 0,C 180,E1 16750.365,E2 16750.365} C_VEL
LIN {X 0,Y 424.984,Z 873.826,A -85,B 0,C 180,E1 16754.847,E2 16754.847} C_VEL
LIN {X 0,Y 430.038,Z 855.532,A -85,B 0,C 180,E1 16759.02,E2 16759.02} C_VEL
LIN {X 0,Y 436.743,Z 831.181,A -85,B 0,C 180,E1 16762.884,E2 16762.884} C_VEL
LIN {X 0,Y 445.147,Z 799.654,A -85,B 0,C 180,E1 16766.532,E2 16766.532} C_VEL
LIN {X 0,Y 455.609,Z 760.306,A -85,B 0,C 180,E1 16769.822,E2 16769.822} C_VEL
LIN {X 0,Y 466.686,Z 717.509,A -85,B 0,C 180,E1 16772.305,E2 16772.305} C_VEL
LIN {X 0,Y 472.646,Z 691.543,A -85,B 0,C 180,E1 16773.442,E2 16773.442} C_VEL
LIN {X 0,Y 471.967,Z 682.579,A -85,B 0,C 180,E1 16775.295,E2 16775.295} C_VEL
LIN {X 0,Y 472.569,Z 678.328,A -85,B 0,C 180,E1 16777.62,E2 16777.62} C_VEL
LIN {X 0,Y 474.187,Z 684.409,A -85,B 0,C 180,E1 16779.84,E2 16779.84} C_VEL
LIN {X 0,Y 476.195,Z 694.967,A -85,B 0,C 180,E1 16781.485,E2 16781.485} C_VEL
LIN {X 0,Y 476.732,Z 710.486,A -85,B 0,C 180,E1 16782.773,E2 16782.773} C_VEL
LIN {X 0,Y 467.505,Z 755.926,A -85,B 0,C 180,E1 16784.608,E2 16784.608} C_VEL
LIN {X 0,Y 457.439,Z 798.262,A -85,B 0,C 180,E1 16787.141,E2 16787.141} C_VEL
LIN {X 0,Y 446.51,Z 840.423,A -85,B 0,C 180,E1 16790.65,E2 16790.65} C_VEL
LIN {X 0,Y 436.374,Z 878.08,A -85,B 0,C 180,E1 16794.879,E2 16794.879} C_VEL
LIN {X 0,Y 427.523,Z 912.14,A -85,B 0,C 180,E1 16799.966,E2 16799.966} C_VEL
LIN {X 0,Y 420.873,Z 941.406,A -85,B 0,C 180,E1 16805.832,E2 16805.832} C_VEL
LIN {X 0,Y 417.261,Z 962.178,A -85,B 0,C 180,E1 16811.48,E2 16811.48} C_VEL
LIN {X 0,Y 415.69,Z 977.605,A -85,B 0,C 180,E1 16817.373,E2 16817.373} C_VEL
LIN {X 0,Y 415.377,Z 986.56,A -85,B 0,C 180,E1 16822.671,E2 16822.671} C_VEL
LIN {X 0,Y 415.563,Z 990.703,A -85,B 0,C 180,E1 16827.916,E2 16827.916} C_VEL
LIN {X 0,Y 415.499,Z 990.706,A -85,B 0,C 180,E1 16832.096,E2 16832.096} C_VEL
LIN {X 0,Y 415.355,Z 986.445,A -85,B 0,C 180,E1 16837.341,E2 16837.341} C_VEL
LIN {X 0,Y 415.732,Z 977.373,A -85,B 0,C 180,E1 16842.637,E2 16842.637} C_VEL
LIN {X 0,Y 415.835,Z 975.965,A -85,B 0,C 180,E1 16843.25,E2 16843.25} C_VEL
LIN {X 0,Y 412.326,Z 970.132,A -85,B 0,C 180,E1 16845.485,E2 16845.485} C_VEL
LIN {X 0,Y 409.066,Z 963.513,A -85,B 0,C 180,E1 16847.72,E2 16847.72} C_VEL
LIN {X 0,Y 411.843,Z 945.437,A -85,B 0,C 180,E1 16852.806,E2 16852.806} C_VEL
LIN {X 0,Y 416.964,Z 919.552,A -85,B 0,C 180,E1 16858.197,E2 16858.197} C_VEL
LIN {X 0,Y 423.901,Z 887.345,A -85,B 0,C 180,E1 16863.185,E2 16863.185} C_VEL
LIN {X 0,Y 431.835,Z 851.059,A -85,B 0,C 180,E1 16867.372,E2 16867.372} C_VEL
LIN {X 0,Y 439.748,Z 812.119,A -85,B 0,C 180,E1 16870.719,E2 16870.719} C_VEL
LIN {X 0,Y 447.121,Z 769.173,A -85,B 0,C 180,E1 16873.397,E2 16873.397} C_VEL
